   // sequencer 3: Empty Process
   INITIAL_STEP CheckMachineMode:   // S200, max time T#10S, warning time T#7S
   END_STEP
   TRANSITION Trans145 FROM CheckMachineMode TO WaitAllStoperReset   // T200
      := "AutoProcessControl".Global.K.EmptyPallet;
   END_TRANSITION
   STEP Step153:   // S153, max time T#10S, warning time T#7S
   END_STEP
   TRANSITION Trans163 FROM Step153 TO "CheckMachine Mode_6"   // T163, jump
      := TRUE;
   END_TRANSITION
   STEP "Process Finish_8":   // S244, max time T#10S, warning time T#7S
   END_STEP
   TRANSITION Trans257 FROM "Process Finish_8" TO Step153   // T256
      := TRUE;
   END_TRANSITION
   STEP LoadStop_14:   // S61, max time T#10S, warning time T#7S
   END_STEP
   TRANSITION Trans154 FROM LoadStop_14 TO CheckPalletExist_10   // T175
      := #LoadStop_14.T > t#2S;
   END_TRANSITION
   STEP LoadStop_12:   // S62, max time T#10S, warning time T#7S
   END_STEP
   TRANSITION Trans152 FROM LoadStop_12 TO CheckPalletExist_8   // T169
      := #LoadStop_12.T > t#2S;
   END_TRANSITION
   STEP "CheckMachine Mode_5":   // S158, max time T#10S, warning time T#7S
   END_STEP
   TRANSITION Trans175 FROM "CheckMachine Mode_5" TO LoadStop_13   // T196
      := "AutoProcessControl".Global.K.EmptyPallet;
   END_TRANSITION
   STEP LoadStop_13:   // S63, max time T#10S, warning time T#7S
   END_STEP
   TRANSITION Trans153 FROM LoadStop_13 TO CheckPalletExist_9   // T170
      := #LoadStop_13.T > t#2S;
   END_TRANSITION
   STEP CheckPalletExist_7:   // S64, max time T#10S, warning time T#7S
   END_STEP
   TRANSITION Trans66 FROM CheckPalletExist_7 TO WaitLineMotorReady_7   // T65
      := "K-reservePalletEmptyCheck1" AND (#CheckPalletExist_7.T > t#1000MS);
   END_TRANSITION
   TRANSITION Trans33 FROM CheckPalletExist_7 TO WaitPalletArive_9   // T32
      := NOT "K-reservePalletEmptyCheck1" AND (#CheckPalletExist_7.T > t#1000MS);
   END_TRANSITION
   STEP AriveTimeDelay_8:   // S159, max time T#10S, warning time T#7S
   END_STEP
   TRANSITION Trans151 FROM AriveTimeDelay_8 TO StoperReset_8   // T168
      := #AriveTimeDelay_8.T > t#500MS;
   END_TRANSITION
   STEP WaitLineMotorReady_7:   // S65, max time T#10S, warning time T#7S
   END_STEP
   TRANSITION Trans67 FROM WaitLineMotorReady_7 TO WaitPalletRequestRelease_7   // T66
      := "MotorControl".Dev[15].OutControl.o_Ready;
   END_TRANSITION
   STEP WaitPalletRequestRelease_7:   // S66, max time T#10S, warning time T#7S
   END_STEP
   TRANSITION Trans68 FROM WaitPalletRequestRelease_7 TO StoperRelease_8   // T67
      := NOT "iK-reserveTakeGateDetection";
   END_TRANSITION
   STEP LoadStop_11:   // S160, max time T#10S, warning time T#7S
   END_STEP
   TRANSITION Trans781 FROM LoadStop_11 TO CheckPalletExist_7   // T172
      := #LoadStop_11.T > t#2S;
   END_TRANSITION
   STEP WaitPalletArrveNextPos_7:   // S67, max time T#10S, warning time T#7S
   END_STEP
   TRANSITION Trans65 FROM WaitPalletArrveNextPos_7 TO AriveTimeDelay_8   // T64
      := "iK-reserveTakeGateDetection" OR NOT "AutoProcessControl".Global.K.EmptyPallet;
   END_TRANSITION
   STEP "Process Finish_9":   // S245, max time T#10S, warning time T#7S
   END_STEP
   TRANSITION Trans258 FROM "Process Finish_9" TO "CheckMachine Mode_7"   // T257, jump
      := TRUE;
   END_TRANSITION
   STEP StoperReset_8:   // S161, max time T#10S, warning time T#7S
              S    "ST10Cylinder".Cy[43].Inout.AutoGoHome
              R    "ST10Cylinder".Cy[43].Inout.AutoGoWork
   END_STEP
   TRANSITION Trans782 FROM StoperReset_8 TO "Process Finish_8"   // T173
      := TRUE;
   END_TRANSITION
   STEP StoperRelease_8:   // S162, max time T#10S, warning time T#7S
              R    "ST10Cylinder".Cy[43].Inout.AutoGoHome
              S    "ST10Cylinder".Cy[43].Inout.AutoGoWork
   END_STEP
   TRANSITION Trans783 FROM StoperRelease_8 TO WaitPalletArrveNextPos_7   // T174
      := #StoperRelease_8.T > t#1000MS;
   END_TRANSITION
   STEP CheckPalletExist_8:   // S68, max time T#10S, warning time T#7S
   END_STEP
   TRANSITION Trans70 FROM CheckPalletExist_8 TO WaitLineMotorReady_8   // T69
      := "K-reservePalletEmptyCheck2" AND (#CheckPalletExist_8.T > t#1000MS);
   END_TRANSITION
   TRANSITION Trans156 FROM CheckPalletExist_8 TO WaitPalletArive_6   // T179
      := NOT "K-reservePalletEmptyCheck2" AND (#CheckPalletExist_8.T > t#1000MS);
   END_TRANSITION
   STEP AriveTimeDelay_9:   // S163, max time T#10S, warning time T#7S
   END_STEP
   TRANSITION Trans155 FROM AriveTimeDelay_9 TO StoperReset_9   // T176
      := #AriveTimeDelay_9.T > t#500MS;
   END_TRANSITION
   STEP WaitLineMotorReady_8:   // S69, max time T#10S, warning time T#7S
   END_STEP
   TRANSITION Trans71 FROM WaitLineMotorReady_8 TO WaitPalletRequestRelease_8   // T70
      := "MotorControl".Dev[15].OutControl.o_Ready;
   END_TRANSITION
   STEP WaitPalletRequestRelease_8:   // S70, max time T#10S, warning time T#7S
   END_STEP
   TRANSITION Trans72 FROM WaitPalletRequestRelease_8 TO StoperRelease_9   // T71
      := "AutoProcessControl".Global.K.LoadStopRequestPallet_2;
   END_TRANSITION
   STEP WaitPalletArrveNextPos_8:   // S71, max time T#10S, warning time T#7S
   END_STEP
   TRANSITION Trans69 FROM WaitPalletArrveNextPos_8 TO AriveTimeDelay_9   // T68
      := "K-reservePalletEmptyCheck1";
   END_TRANSITION
   STEP StoperReset_9:   // S164, max time T#10S, warning time T#7S
              S    "ST10Cylinder".Cy[44].Inout.AutoGoHome
              R    "ST10Cylinder".Cy[44].Inout.AutoGoWork
   END_STEP
   TRANSITION Trans784 FROM StoperReset_9 TO "Process Finish_9"   // T177
      := TRUE;
   END_TRANSITION
   STEP StoperRelease_9:   // S165, max time T#10S, warning time T#7S
              R    "ST10Cylinder".Cy[44].Inout.AutoGoHome
              S    "ST10Cylinder".Cy[44].Inout.AutoGoWork
   END_STEP
   TRANSITION Trans785 FROM StoperRelease_9 TO WaitPalletArrveNextPos_8   // T178
      := #StoperRelease_9.T > t#1000MS;
   END_TRANSITION
   STEP WaitPalletArive_6:   // S166, max time T#10S, warning time T#7S
              N    "AutoProcessControl".Global.K.LoadStopRequestPallet_3
   END_STEP
   TRANSITION Trans157 FROM WaitPalletArive_6 TO TimeDelay_6   // T180
      := "K-reservePalletEmptyCheck2" OR NOT "AutoProcessControl".Global.K.EmptyPallet;
   END_TRANSITION
   STEP TimeDelay_6:   // S167, max time T#10S, warning time T#7S
   END_STEP
   TRANSITION Trans158 FROM TimeDelay_6 TO "CheckMachine Mode_7"   // T181, jump
      := #TimeDelay_6.T > t#500MS;
   END_TRANSITION
   STEP "Process Finish_10":   // S246, max time T#10S, warning time T#7S
   END_STEP
   TRANSITION Trans259 FROM "Process Finish_10" TO "CheckMachine Mode_5"   // T258, jump
      := TRUE;
   END_TRANSITION
   STEP CheckPalletExist_9:   // S72, max time T#10S, warning time T#7S
   END_STEP
   TRANSITION Trans74 FROM CheckPalletExist_9 TO WaitLineMotorReady_9   // T73
      := "K-reservePalletEmptyCheck3" AND (#CheckPalletExist_9.T > t#1000MS);
   END_TRANSITION
   TRANSITION Trans160 FROM CheckPalletExist_9 TO WaitPalletArive_7   // T185
      := NOT "K-reservePalletEmptyCheck3" AND (#CheckPalletExist_9.T > t#1000MS);
   END_TRANSITION
   STEP AriveTimeDelay_10:   // S168, max time T#10S, warning time T#7S
   END_STEP
   TRANSITION Trans159 FROM AriveTimeDelay_10 TO StoperReset_10   // T182
      := #AriveTimeDelay_10.T > t#500MS;
   END_TRANSITION
   STEP WaitLineMotorReady_9:   // S73, max time T#10S, warning time T#7S
   END_STEP
   TRANSITION Trans75 FROM WaitLineMotorReady_9 TO WaitPalletRequestRelease_9   // T74
      := "MotorControl".Dev[15].OutControl.o_Ready;
   END_TRANSITION
   STEP WaitPalletRequestRelease_9:   // S74, max time T#10S, warning time T#7S
   END_STEP
   TRANSITION Trans76 FROM WaitPalletRequestRelease_9 TO StoperRelease_10   // T75
      := "AutoProcessControl".Global.K.LoadStopRequestPallet_3;
   END_TRANSITION
   STEP WaitPalletArrveNextPos_9:   // S75, max time T#10S, warning time T#7S
   END_STEP
   TRANSITION Trans73 FROM WaitPalletArrveNextPos_9 TO AriveTimeDelay_10   // T72
      := "K-reservePalletEmptyCheck2";
   END_TRANSITION
   STEP StoperReset_10:   // S169, max time T#10S, warning time T#7S
              S    "ST10Cylinder".Cy[45].Inout.AutoGoHome
              R    "ST10Cylinder".Cy[45].Inout.AutoGoWork
   END_STEP
   TRANSITION Trans786 FROM StoperReset_10 TO "Process Finish_10"   // T183
      := TRUE;
   END_TRANSITION
   STEP StoperRelease_10:   // S170, max time T#10S, warning time T#7S
              R    "ST10Cylinder".Cy[45].Inout.AutoGoHome
              S    "ST10Cylinder".Cy[45].Inout.AutoGoWork
   END_STEP
   TRANSITION Trans787 FROM StoperRelease_10 TO WaitPalletArrveNextPos_9   // T184
      := #StoperRelease_10.T > t#1000MS;
   END_TRANSITION
   STEP WaitPalletArive_7:   // S171, max time T#10S, warning time T#7S
              N    "AutoProcessControl".Global.K.LoadStopRequestPallet_4
   END_STEP
   TRANSITION Trans161 FROM WaitPalletArive_7 TO TimeDelay_7   // T186
      := "K-reservePalletEmptyCheck3" OR NOT "AutoProcessControl".Global.K.EmptyPallet;
   END_TRANSITION
   STEP TimeDelay_7:   // S172, max time T#10S, warning time T#7S
   END_STEP
   TRANSITION Trans162 FROM TimeDelay_7 TO "CheckMachine Mode_5"   // T187, jump
      := #TimeDelay_7.T > t#500MS;
   END_TRANSITION
   STEP "Process Finish_11":   // S247, max time T#10S, warning time T#7S
   END_STEP
   TRANSITION Trans260 FROM "Process Finish_11" TO "CheckMachine Mode_8"   // T259, jump
      := TRUE;
   END_TRANSITION
   STEP CheckPalletExist_10:   // S76, max time T#10S, warning time T#7S
   END_STEP
   TRANSITION Trans78 FROM CheckPalletExist_10 TO WaitLineMotorReady_10   // T77
      := "K-reservePalletEmptyCheck4" AND NOT "iK-reserveMiddleDetection" AND (#CheckPalletExist_10.T > t#1000MS);
   END_TRANSITION
   TRANSITION Trans170 FROM CheckPalletExist_10 TO WaitPalletArive_8   // T191
      := NOT "K-reservePalletEmptyCheck4" AND (#CheckPalletExist_10.T > t#1000MS);
   END_TRANSITION
   STEP AriveTimeDelay_11:   // S173, max time T#10S, warning time T#7S
   END_STEP
   TRANSITION Trans169 FROM AriveTimeDelay_11 TO StoperReset_11   // T188
      := #AriveTimeDelay_11.T > t#500MS;
   END_TRANSITION
   STEP WaitLineMotorReady_10:   // S77, max time T#10S, warning time T#7S
   END_STEP
   TRANSITION Trans79 FROM WaitLineMotorReady_10 TO WaitPalletRequestRelease_10   // T78
      := "MotorControl".Dev[15].OutControl.o_Ready;
   END_TRANSITION
   STEP WaitPalletRequestRelease_10:   // S78, max time T#10S, warning time T#7S
   END_STEP
   TRANSITION Trans80 FROM WaitPalletRequestRelease_10 TO StoperRelease_11   // T79
      := "AutoProcessControl".Global.K.LoadStopRequestPallet_4;
   END_TRANSITION
   STEP WaitPalletArrveNextPos_10:   // S79, max time T#10S, warning time T#7S
   END_STEP
   TRANSITION Trans77 FROM WaitPalletArrveNextPos_10 TO AriveTimeDelay_11   // T76
      := "K-reservePalletEmptyCheck3";
   END_TRANSITION
   STEP StoperReset_11:   // S174, max time T#10S, warning time T#7S
              S    "ST10Cylinder".Cy[46].Inout.AutoGoHome
              R    "ST10Cylinder".Cy[46].Inout.AutoGoWork
   END_STEP
   TRANSITION Trans788 FROM StoperReset_11 TO "Process Finish_11"   // T189
      := TRUE;
   END_TRANSITION
   STEP StoperRelease_11:   // S175, max time T#10S, warning time T#7S
              R    "ST10Cylinder".Cy[46].Inout.AutoGoHome
              S    "ST10Cylinder".Cy[46].Inout.AutoGoWork
   END_STEP
   TRANSITION Trans789 FROM StoperRelease_11 TO WaitPalletArrveNextPos_10   // T190
      := #StoperRelease_11.T > t#1000MS;
   END_TRANSITION
   STEP WaitPalletArive_8:   // S176, max time T#10S, warning time T#7S
   END_STEP
   TRANSITION Trans171 FROM WaitPalletArive_8 TO TimeDelay_8   // T192
      := ("K-reservePalletEmptyCheck4" AND NOT "iK-reserveMiddleDetection") OR NOT "AutoProcessControl".Global.K.EmptyPallet;
   END_TRANSITION
   STEP TimeDelay_8:   // S177, max time T#10S, warning time T#7S
   END_STEP
   TRANSITION Trans172 FROM TimeDelay_8 TO "CheckMachine Mode_8"   // T193, jump
      := #TimeDelay_8.T > t#500MS;
   END_TRANSITION
   STEP "CheckMachine Mode_6":   // S178, max time T#10S, warning time T#7S
   END_STEP
   TRANSITION Trans173 FROM "CheckMachine Mode_6" TO LoadStop_11   // T194
      := "AutoProcessControl".Global.K.EmptyPallet;
   END_TRANSITION
   STEP "CheckMachine Mode_7":   // S179, max time T#10S, warning time T#7S
   END_STEP
   TRANSITION Trans174 FROM "CheckMachine Mode_7" TO LoadStop_12   // T195
      := "AutoProcessControl".Global.K.EmptyPallet;
   END_TRANSITION
   STEP "CheckMachine Mode_8":   // S180, max time T#10S, warning time T#7S
   END_STEP
   TRANSITION Trans168 FROM "CheckMachine Mode_8" TO LoadStop_14   // T171
      := "AutoProcessControl".Global.K.EmptyPallet;
   END_TRANSITION
   STEP WaitAllStoperReset:   // S181, max time T#10S, warning time T#7S
   END_STEP
   TRANSITION Trans197 FROM WaitAllStoperReset TO MotorRun_1   // T197
      := "ST10Cylinder".Cy[43].Inout.AutoGoHome AND NOT "ST10Cylinder".Cy[43].Inout.AutoGoWork AND "ST10Cylinder".Cy[44].Inout.AutoGoHome AND NOT "ST10Cylinder".Cy[44].Inout.AutoGoWork AND "ST10Cylinder".Cy[45].Inout.AutoGoHome AND NOT "ST10Cylinder".Cy[45].Inout.AutoGoWork AND "ST10Cylinder".Cy[46].Inout.AutoGoHome AND NOT "ST10Cylinder".Cy[46].Inout.AutoGoWork;
   END_TRANSITION
   STEP Step182:   // S182, max time T#10S, warning time T#7S
   END_STEP
   TRANSITION Trans198 FROM Step182 TO ("CheckMachine Mode_7", "CheckMachine Mode_5", "CheckMachine Mode_8", "CheckMachine Mode_6")   // T198
      := TRUE;
   END_TRANSITION
   STEP MotorRun_1:   // S80, max time T#10S, warning time T#7S
              R    "MotorControl".Dev[15].Auto.Start
              S    "MotorControl".Dev[15].Auto.CCWStart
              S    "MotorControl".Dev[16].Auto.Start
              R    "MotorControl".Dev[16].Auto.CCWStart
   END_STEP
   TRANSITION Trans81 FROM MotorRun_1 TO Step182   // T80
      := TRUE;
   END_TRANSITION
   STEP WaitPalletArive_9:   // S183, max time T#10S, warning time T#7S
              N    "AutoProcessControl".Global.K.LoadStopRequestPallet_2
   END_STEP
   TRANSITION Trans176 FROM WaitPalletArive_9 TO TimeDelay_9   // T199
      := "K-reservePalletEmptyCheck1" OR NOT "AutoProcessControl".Global.K.EmptyPallet;
   END_TRANSITION
   STEP TimeDelay_9:   // S184, max time T#10S, warning time T#7S
   END_STEP
   TRANSITION Trans177 FROM TimeDelay_9 TO "CheckMachine Mode_6"   // T201, jump
      := #TimeDelay_9.T > t#500MS;
   END_TRANSITION

   // permanent post-instructions
   NETWORK 1
      #ioPM_Inface.StepNum := #RT_DATA.S_DISPLAY;
   NETWORK 2
      IF #iSysInface.Reset THEN #AlarmID := 0; END_IF;
   NETWORK 3
      #TON[10].TON(IN := #工件放行中, PT := T#0.5S);
      IF #TON[10].Q THEN #工件放行中 := FALSE; END_IF;
END_FUNCTION_BLOCK

FUNCTION "ST10Cyl_interface91-100" : Void   // FC1029, LAD
{ S7_Optimized_Access := 'FALSE' }
// stored: AutoNumber false, SetENOAutomatically false
   VAR_INPUT
      AlwaysON : Bool;
      E_stop : Bool;
   END_VAR
   VAR_TEMP
      tTest : Bool;
   END_VAR
BEGIN

REGION Network 1 (SCL): Cylinder 91-100 IO Interface (SCL)
END_REGION

REGION Network 2: CY91 interface
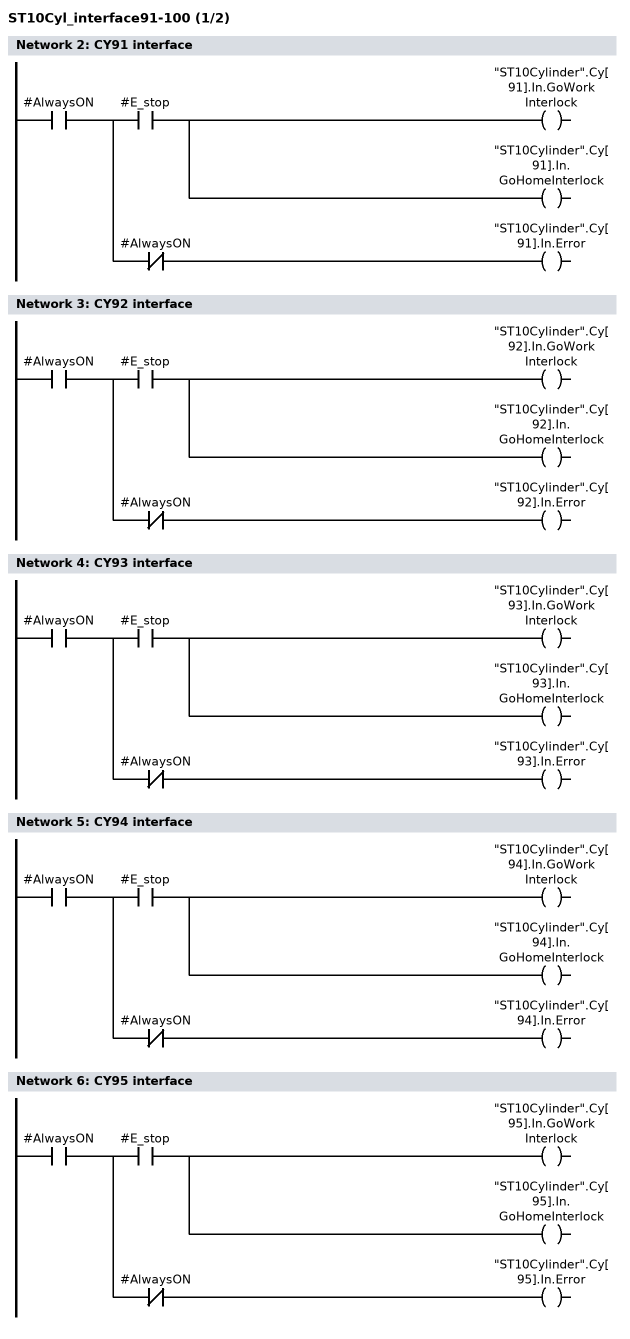
   RUNG wire#powerrail
      Contact( #AlwaysON )
      wire#w1
      Contact( #E_stop )
      wire#w2
      Coil( "ST10Cylinder".Cy[91].In.GoWorkInterlock )
   END_RUNG
   RUNG wire#w2
      Coil( "ST10Cylinder".Cy[91].In.GoHomeInterlock )
   END_RUNG
   RUNG wire#w1
      I_Contact( #AlwaysON )
      Coil( "ST10Cylinder".Cy[91].In.Error )
   END_RUNG
   // the same network as SCL:
   "ST10Cylinder".Cy[91].In.GoWorkInterlock := #AlwaysON AND #E_stop;
   "ST10Cylinder".Cy[91].In.GoHomeInterlock := #AlwaysON AND #E_stop;
   "ST10Cylinder".Cy[91].In.Error := #AlwaysON AND NOT #AlwaysON;
END_REGION

REGION Network 3: CY92 interface
   RUNG wire#powerrail
      Contact( #AlwaysON )
      wire#w1
      Contact( #E_stop )
      wire#w2
      Coil( "ST10Cylinder".Cy[92].In.GoWorkInterlock )
   END_RUNG
   RUNG wire#w2
      Coil( "ST10Cylinder".Cy[92].In.GoHomeInterlock )
   END_RUNG
   RUNG wire#w1
      I_Contact( #AlwaysON )
      Coil( "ST10Cylinder".Cy[92].In.Error )
   END_RUNG
   // the same network as SCL:
   "ST10Cylinder".Cy[92].In.GoWorkInterlock := #AlwaysON AND #E_stop;
   "ST10Cylinder".Cy[92].In.GoHomeInterlock := #AlwaysON AND #E_stop;
   "ST10Cylinder".Cy[92].In.Error := #AlwaysON AND NOT #AlwaysON;
END_REGION

REGION Network 4: CY93 interface
   RUNG wire#powerrail
      Contact( #AlwaysON )
      wire#w1
      Contact( #E_stop )
      wire#w2
      Coil( "ST10Cylinder".Cy[93].In.GoWorkInterlock )
   END_RUNG
   RUNG wire#w2
      Coil( "ST10Cylinder".Cy[93].In.GoHomeInterlock )
   END_RUNG
   RUNG wire#w1
      I_Contact( #AlwaysON )
      Coil( "ST10Cylinder".Cy[93].In.Error )
   END_RUNG
   // the same network as SCL:
   "ST10Cylinder".Cy[93].In.GoWorkInterlock := #AlwaysON AND #E_stop;
   "ST10Cylinder".Cy[93].In.GoHomeInterlock := #AlwaysON AND #E_stop;
   "ST10Cylinder".Cy[93].In.Error := #AlwaysON AND NOT #AlwaysON;
END_REGION

REGION Network 5: CY94 interface
   RUNG wire#powerrail
      Contact( #AlwaysON )
      wire#w1
      Contact( #E_stop )
      wire#w2
      Coil( "ST10Cylinder".Cy[94].In.GoWorkInterlock )
   END_RUNG
   RUNG wire#w2
      Coil( "ST10Cylinder".Cy[94].In.GoHomeInterlock )
   END_RUNG
   RUNG wire#w1
      I_Contact( #AlwaysON )
      Coil( "ST10Cylinder".Cy[94].In.Error )
   END_RUNG
   // the same network as SCL:
   "ST10Cylinder".Cy[94].In.GoWorkInterlock := #AlwaysON AND #E_stop;
   "ST10Cylinder".Cy[94].In.GoHomeInterlock := #AlwaysON AND #E_stop;
   "ST10Cylinder".Cy[94].In.Error := #AlwaysON AND NOT #AlwaysON;
END_REGION

REGION Network 6: CY95 interface
   RUNG wire#powerrail
      Contact( #AlwaysON )
      wire#w1
      Contact( #E_stop )
      wire#w2
      Coil( "ST10Cylinder".Cy[95].In.GoWorkInterlock )
   END_RUNG
   RUNG wire#w2
      Coil( "ST10Cylinder".Cy[95].In.GoHomeInterlock )
   END_RUNG
   RUNG wire#w1
      I_Contact( #AlwaysON )
      Coil( "ST10Cylinder".Cy[95].In.Error )
   END_RUNG
   // the same network as SCL:
   "ST10Cylinder".Cy[95].In.GoWorkInterlock := #AlwaysON AND #E_stop;
   "ST10Cylinder".Cy[95].In.GoHomeInterlock := #AlwaysON AND #E_stop;
   "ST10Cylinder".Cy[95].In.Error := #AlwaysON AND NOT #AlwaysON;
END_REGION

REGION Network 7: CY96 interface
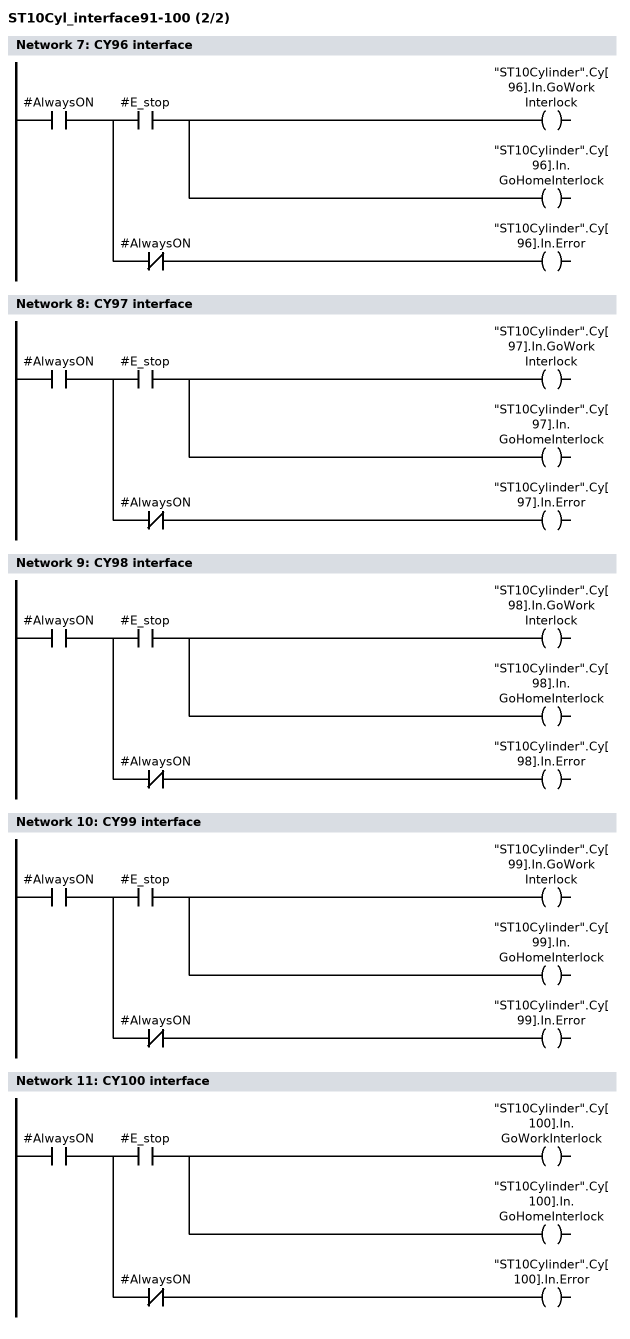
   RUNG wire#powerrail
      Contact( #AlwaysON )
      wire#w1
      Contact( #E_stop )
      wire#w2
      Coil( "ST10Cylinder".Cy[96].In.GoWorkInterlock )
   END_RUNG
   RUNG wire#w2
      Coil( "ST10Cylinder".Cy[96].In.GoHomeInterlock )
   END_RUNG
   RUNG wire#w1
      I_Contact( #AlwaysON )
      Coil( "ST10Cylinder".Cy[96].In.Error )
   END_RUNG
   // the same network as SCL:
   "ST10Cylinder".Cy[96].In.GoWorkInterlock := #AlwaysON AND #E_stop;
   "ST10Cylinder".Cy[96].In.GoHomeInterlock := #AlwaysON AND #E_stop;
   "ST10Cylinder".Cy[96].In.Error := #AlwaysON AND NOT #AlwaysON;
END_REGION

REGION Network 8: CY97 interface
   RUNG wire#powerrail
      Contact( #AlwaysON )
      wire#w1
      Contact( #E_stop )
      wire#w2
      Coil( "ST10Cylinder".Cy[97].In.GoWorkInterlock )
   END_RUNG
   RUNG wire#w2
      Coil( "ST10Cylinder".Cy[97].In.GoHomeInterlock )
   END_RUNG
   RUNG wire#w1
      I_Contact( #AlwaysON )
      Coil( "ST10Cylinder".Cy[97].In.Error )
   END_RUNG
   // the same network as SCL:
   "ST10Cylinder".Cy[97].In.GoWorkInterlock := #AlwaysON AND #E_stop;
   "ST10Cylinder".Cy[97].In.GoHomeInterlock := #AlwaysON AND #E_stop;
   "ST10Cylinder".Cy[97].In.Error := #AlwaysON AND NOT #AlwaysON;
END_REGION

REGION Network 9: CY98 interface
   RUNG wire#powerrail
      Contact( #AlwaysON )
      wire#w1
      Contact( #E_stop )
      wire#w2
      Coil( "ST10Cylinder".Cy[98].In.GoWorkInterlock )
   END_RUNG
   RUNG wire#w2
      Coil( "ST10Cylinder".Cy[98].In.GoHomeInterlock )
   END_RUNG
   RUNG wire#w1
      I_Contact( #AlwaysON )
      Coil( "ST10Cylinder".Cy[98].In.Error )
   END_RUNG
   // the same network as SCL:
   "ST10Cylinder".Cy[98].In.GoWorkInterlock := #AlwaysON AND #E_stop;
   "ST10Cylinder".Cy[98].In.GoHomeInterlock := #AlwaysON AND #E_stop;
   "ST10Cylinder".Cy[98].In.Error := #AlwaysON AND NOT #AlwaysON;
END_REGION

REGION Network 10: CY99 interface
   RUNG wire#powerrail
      Contact( #AlwaysON )
      wire#w1
      Contact( #E_stop )
      wire#w2
      Coil( "ST10Cylinder".Cy[99].In.GoWorkInterlock )
   END_RUNG
   RUNG wire#w2
      Coil( "ST10Cylinder".Cy[99].In.GoHomeInterlock )
   END_RUNG
   RUNG wire#w1
      I_Contact( #AlwaysON )
      Coil( "ST10Cylinder".Cy[99].In.Error )
   END_RUNG
   // the same network as SCL:
   "ST10Cylinder".Cy[99].In.GoWorkInterlock := #AlwaysON AND #E_stop;
   "ST10Cylinder".Cy[99].In.GoHomeInterlock := #AlwaysON AND #E_stop;
   "ST10Cylinder".Cy[99].In.Error := #AlwaysON AND NOT #AlwaysON;
END_REGION

REGION Network 11: CY100 interface
   RUNG wire#powerrail
      Contact( #AlwaysON )
      wire#w1
      Contact( #E_stop )
      wire#w2
      Coil( "ST10Cylinder".Cy[100].In.GoWorkInterlock )
   END_RUNG
   RUNG wire#w2
      Coil( "ST10Cylinder".Cy[100].In.GoHomeInterlock )
   END_RUNG
   RUNG wire#w1
      I_Contact( #AlwaysON )
      Coil( "ST10Cylinder".Cy[100].In.Error )
   END_RUNG
   // the same network as SCL:
   "ST10Cylinder".Cy[100].In.GoWorkInterlock := #AlwaysON AND #E_stop;
   "ST10Cylinder".Cy[100].In.GoHomeInterlock := #AlwaysON AND #E_stop;
   "ST10Cylinder".Cy[100].In.Error := #AlwaysON AND NOT #AlwaysON;
END_REGION
END_FUNCTION

FUNCTION_BLOCK "ST10_Stopper_FB"   // FB1160, LAD
{ S7_Optimized_Access := 'TRUE' }
// stored: AutoNumber false, MemoryReserve 100, SetENOAutomatically false
   VAR
      FB_Stopper_Instance { S7_SetPoint := 'True'} : Array[1..3] of "FB_Stopper";
   END_VAR
BEGIN

REGION Network 1 (SCL): A-托盘缓存阻挡气缸
       (*  
       REGION 允许释放条件,根据实际完善
           //马达运行中且工位一允许进料
           IF "ST350_Motor_InterfaceDB".aDev[1].Run  THEN
               "ST350_Stopper_InterfaceDB".Command[1].In.iReleaseClear := TRUE;
           ELSE
               "ST350_Stopper_InterfaceDB".Command[1].In.iReleaseClear := FALSE;
           END_IF;
       END_REGION

       REGION IO_image
           //InPut
           "ST350_Stopper_InterfaceDB".Command[1].In.iSensor := "iBurfferPalletDetection";//本站托盘到位
           "ST350_Stopper_InterfaceDB".Command[1].In.iNextSensor := "iWork01PalletDetection";//后站托盘到位
           "ST350_Stopper_InterfaceDB".Command[1].In.iNextValve := "oA-Lifting-01StopperCylinder";//后站挡停输出

           // //OutPut
            "ST10Cylinder".Cy[5].Inout.AutoGoWork:= "ST350_Stopper_InterfaceDB".Command[1].Out.oValve;//本站挡停输出
       END_REGION


       *)
END_REGION

REGION Network 2: #FB_Stopper_Instance[1] A-托盘缓存阻挡气缸
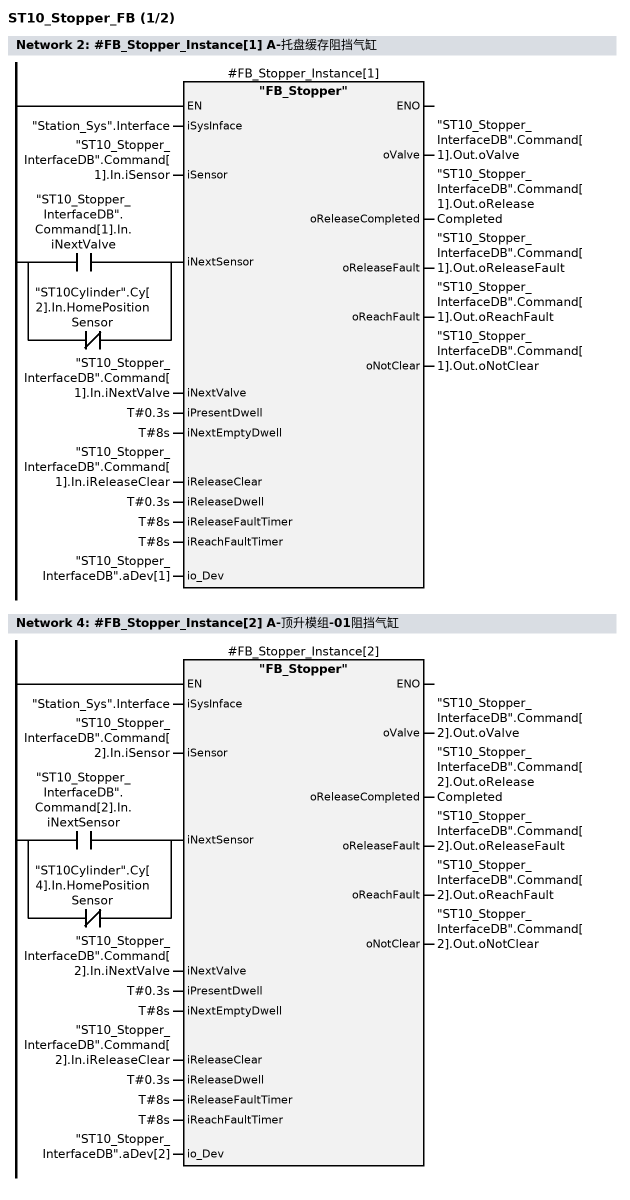
   RUNG wire#powerrail
      #FB_Stopper_Instance[1](iNextSensor := wire#w1, iSysInface := "Station_Sys".Interface, iSensor := "ST10_Stopper_InterfaceDB".Command[1].In.iSensor, iNextValve := "ST10_Stopper_InterfaceDB".Command[1].In.iNextValve, iPresentDwell := T#0.3s, iNextEmptyDwell := T#8s, iReleaseClear := "ST10_Stopper_InterfaceDB".Command[1].In.iReleaseClear, iReleaseDwell := T#0.3s, iReleaseFaultTimer := T#8s, iReachFaultTimer := T#8s, io_Dev := "ST10_Stopper_InterfaceDB".aDev[1], oValve => "ST10_Stopper_InterfaceDB".Command[1].Out.oValve, oReleaseCompleted => "ST10_Stopper_InterfaceDB".Command[1].Out.oReleaseCompleted, oReleaseFault => "ST10_Stopper_InterfaceDB".Command[1].Out.oReleaseFault, oReachFault => "ST10_Stopper_InterfaceDB".Command[1].Out.oReachFault, oNotClear => "ST10_Stopper_InterfaceDB".Command[1].Out.oNotClear)
   END_RUNG
   RUNG wire#powerrail
      Contact( "ST10_Stopper_InterfaceDB".Command[1].In.iNextValve )
   END_RUNG wire#w1
   RUNG wire#powerrail
      I_Contact( "ST10Cylinder".Cy[2].In.HomePositionSensor )
   END_RUNG wire#w1
   // the same network as SCL:
   #FB_Stopper_Instance[1](iSysInface := "Station_Sys".Interface,   // "FB_Stopper"
                           iSensor := "ST10_Stopper_InterfaceDB".Command[1].In.iSensor,
                           iNextSensor := "ST10_Stopper_InterfaceDB".Command[1].In.iNextValve OR NOT "ST10Cylinder".Cy[2].In.HomePositionSensor,
                           iNextValve := "ST10_Stopper_InterfaceDB".Command[1].In.iNextValve,
                           iPresentDwell := T#0.3s,
                           iNextEmptyDwell := T#8s,
                           iReleaseClear := "ST10_Stopper_InterfaceDB".Command[1].In.iReleaseClear,
                           iReleaseDwell := T#0.3s,
                           iReleaseFaultTimer := T#8s,
                           iReachFaultTimer := T#8s,
                           io_Dev := "ST10_Stopper_InterfaceDB".aDev[1],
                           oValve => "ST10_Stopper_InterfaceDB".Command[1].Out.oValve,
                           oReleaseCompleted => "ST10_Stopper_InterfaceDB".Command[1].Out.oReleaseCompleted,
                           oReleaseFault => "ST10_Stopper_InterfaceDB".Command[1].Out.oReleaseFault,
                           oReachFault => "ST10_Stopper_InterfaceDB".Command[1].Out.oReachFault,
                           oNotClear => "ST10_Stopper_InterfaceDB".Command[1].Out.oNotClear);
END_REGION

REGION Network 3 (SCL): A-顶升模组-01阻挡气缸
   (*
   REGION 允许释放条件,根据实际完善:顶升下降且线体运行中
       IF "ST10Cylinder".Cy[2].In.HomePositionSensor AND ("ST350_Motor_InterfaceDB".aDev[1].Run OR "Station_Sys".Manual.Mode) THEN//
           "ST350_Stopper_InterfaceDB".Command[2].In.iReleaseClear := True;
       ELSE
           "ST350_Stopper_InterfaceDB".Command[2].In.iReleaseClear := FALSE;
       END_IF;
   END_REGION

   REGION IO_image
       //InPut
       "ST350_Stopper_InterfaceDB".Command[2].In.iSensor := "iWork01PalletDetection";//本站托盘到位
       "ST350_Stopper_InterfaceDB".Command[2].In.iNextSensor := "iWork02PalletDetection";//后站托盘到位
       "ST350_Stopper_InterfaceDB".Command[2].In.iNextValve := "oA-Lifting-02StopperCylinder";//后站挡停输出

       // //OutPut
        "ST10Cylinder".Cy[1].Inout.AutoGoWork:= "ST350_Stopper_InterfaceDB".Command[2].Out.oValve;//本站挡停输出
   END_REGION

   *0
END_REGION

REGION Network 4: #FB_Stopper_Instance[2] A-顶升模组-01阻挡气缸
   RUNG wire#powerrail
      #FB_Stopper_Instance[2](iNextSensor := wire#w1, iSysInface := "Station_Sys".Interface, iSensor := "ST10_Stopper_InterfaceDB".Command[2].In.iSensor, iNextValve := "ST10_Stopper_InterfaceDB".Command[2].In.iNextValve, iPresentDwell := T#0.3s, iNextEmptyDwell := T#8s, iReleaseClear := "ST10_Stopper_InterfaceDB".Command[2].In.iReleaseClear, iReleaseDwell := T#0.3s, iReleaseFaultTimer := T#8s, iReachFaultTimer := T#8s, io_Dev := "ST10_Stopper_InterfaceDB".aDev[2], oValve => "ST10_Stopper_InterfaceDB".Command[2].Out.oValve, oReleaseCompleted => "ST10_Stopper_InterfaceDB".Command[2].Out.oReleaseCompleted, oReleaseFault => "ST10_Stopper_InterfaceDB".Command[2].Out.oReleaseFault, oReachFault => "ST10_Stopper_InterfaceDB".Command[2].Out.oReachFault, oNotClear => "ST10_Stopper_InterfaceDB".Command[2].Out.oNotClear)
   END_RUNG
   RUNG wire#powerrail
      Contact( "ST10_Stopper_InterfaceDB".Command[2].In.iNextSensor )
   END_RUNG wire#w1
   RUNG wire#powerrail
      I_Contact( "ST10Cylinder".Cy[4].In.HomePositionSensor )
   END_RUNG wire#w1
   // the same network as SCL:
   #FB_Stopper_Instance[2](iSysInface := "Station_Sys".Interface,   // "FB_Stopper"
                           iSensor := "ST10_Stopper_InterfaceDB".Command[2].In.iSensor,
                           iNextSensor := "ST10_Stopper_InterfaceDB".Command[2].In.iNextSensor OR NOT "ST10Cylinder".Cy[4].In.HomePositionSensor,
                           iNextValve := "ST10_Stopper_InterfaceDB".Command[2].In.iNextValve,
                           iPresentDwell := T#0.3s,
                           iNextEmptyDwell := T#8s,
                           iReleaseClear := "ST10_Stopper_InterfaceDB".Command[2].In.iReleaseClear,
                           iReleaseDwell := T#0.3s,
                           iReleaseFaultTimer := T#8s,
                           iReachFaultTimer := T#8s,
                           io_Dev := "ST10_Stopper_InterfaceDB".aDev[2],
                           oValve => "ST10_Stopper_InterfaceDB".Command[2].Out.oValve,
                           oReleaseCompleted => "ST10_Stopper_InterfaceDB".Command[2].Out.oReleaseCompleted,
                           oReleaseFault => "ST10_Stopper_InterfaceDB".Command[2].Out.oReleaseFault,
                           oReachFault => "ST10_Stopper_InterfaceDB".Command[2].Out.oReachFault,
                           oNotClear => "ST10_Stopper_InterfaceDB".Command[2].Out.oNotClear);
END_REGION

REGION Network 5 (SCL): A-顶升模组-02阻挡气缸
   //允许释放条件,根据实际完善:顶升下降且线体运行中
   (*

   REGION IOimage
       //InPut
       "ST350_Stopper_InterfaceDB".Command[3].In.iSensor := "iWork02PalletDetection";//本站托盘到位
       "ST350_Stopper_InterfaceDB".Command[3].In.iNextSensor := "iD-LiftingDetection" AND NOT "iD-LiftingINDetection" ;//后站托盘到位

       //替换后站挡停释放信号：升降机在下&顶升下&无料&允许金托盘
       // "ST350_Stopper_InterfaceDB".Command[3].In.iNextValve := ;//后站挡停输出

       // //OutPut
        "ST10Cylinder".Cy[3].Inout.AutoGoWork := "ST350_Stopper_InterfaceDB".Command[3].Out.oValve;//本站挡停输出


   END_REGION

   *)
END_REGION

REGION Network 6: #FB_Stopper_Instance[3] A-顶升模组-02阻挡气缸
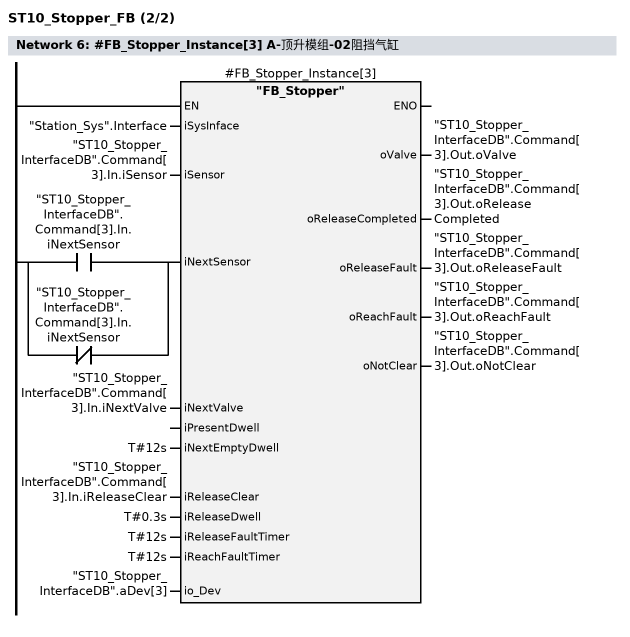
   RUNG wire#powerrail
      #FB_Stopper_Instance[3](iNextSensor := wire#w1, iSysInface := "Station_Sys".Interface, iSensor := "ST10_Stopper_InterfaceDB".Command[3].In.iSensor, iNextValve := "ST10_Stopper_InterfaceDB".Command[3].In.iNextValve, iPresentDwell :=, iNextEmptyDwell := T#12s, iReleaseClear := "ST10_Stopper_InterfaceDB".Command[3].In.iReleaseClear, iReleaseDwell := T#0.3s, iReleaseFaultTimer := T#12s, iReachFaultTimer := T#12s, io_Dev := "ST10_Stopper_InterfaceDB".aDev[3], oValve => "ST10_Stopper_InterfaceDB".Command[3].Out.oValve, oReleaseCompleted => "ST10_Stopper_InterfaceDB".Command[3].Out.oReleaseCompleted, oReleaseFault => "ST10_Stopper_InterfaceDB".Command[3].Out.oReleaseFault, oReachFault => "ST10_Stopper_InterfaceDB".Command[3].Out.oReachFault, oNotClear => "ST10_Stopper_InterfaceDB".Command[3].Out.oNotClear)
   END_RUNG
   RUNG wire#powerrail
      Contact( "ST10_Stopper_InterfaceDB".Command[3].In.iNextSensor )
   END_RUNG wire#w1
   RUNG wire#powerrail
      I_Contact( "ST10_Stopper_InterfaceDB".Command[3].In.iNextSensor )
   END_RUNG wire#w1
   // the same network as SCL:
   #FB_Stopper_Instance[3](iSysInface := "Station_Sys".Interface,   // "FB_Stopper"
                           iSensor := "ST10_Stopper_InterfaceDB".Command[3].In.iSensor,
                           iNextSensor := "ST10_Stopper_InterfaceDB".Command[3].In.iNextSensor OR NOT "ST10_Stopper_InterfaceDB".Command[3].In.iNextSensor,
                           iNextValve := "ST10_Stopper_InterfaceDB".Command[3].In.iNextValve,
                           iNextEmptyDwell := T#12s,
                           iReleaseClear := "ST10_Stopper_InterfaceDB".Command[3].In.iReleaseClear,
                           iReleaseDwell := T#0.3s,
                           iReleaseFaultTimer := T#12s,
                           iReachFaultTimer := T#12s,
                           io_Dev := "ST10_Stopper_InterfaceDB".aDev[3],
                           oValve => "ST10_Stopper_InterfaceDB".Command[3].Out.oValve,
                           oReleaseCompleted => "ST10_Stopper_InterfaceDB".Command[3].Out.oReleaseCompleted,
                           oReleaseFault => "ST10_Stopper_InterfaceDB".Command[3].Out.oReleaseFault,
                           oReachFault => "ST10_Stopper_InterfaceDB".Command[3].Out.oReachFault,
                           oNotClear => "ST10_Stopper_InterfaceDB".Command[3].Out.oNotClear);
END_REGION
END_FUNCTION_BLOCK

FUNCTION_BLOCK "SevroStart&PosCheck"   // FB4073, LAD
{ S7_Optimized_Access := 'TRUE' }
// stored: AutoNumber false, MemoryReserve 100, SetENOAutomatically false
   VAR_INPUT
      iRef_Homed { ExternalAccessible := 'False'; ExternalVisible := 'False'; ExternalWritable := 'False'} : Bool;
      iStandstill { ExternalAccessible := 'False'; ExternalVisible := 'False'; ExternalWritable := 'False'} : Bool;
      iReset : Bool;
      interlcok : Bool;   // 启动互锁
      "iActual Posi" { ExternalAccessible := 'False'; ExternalVisible := 'False'; ExternalWritable := 'False'} : DInt;
      "iTol+" { ExternalAccessible := 'False'; ExternalVisible := 'False'; ExternalWritable := 'False'} : DInt;
      "iTol-" { ExternalAccessible := 'False'; ExternalVisible := 'False'; ExternalWritable := 'False'} : DInt;
      iStartTon : Time := T#200ms;   // 启动延迟
   END_VAR
   VAR_OUTPUT
      oStartPos : Bool;   // 启动
      DoublePosError : Bool;   // 多位置触发
   END_VAR
   VAR_IN_OUT
      ioPoint : Array[0..39] of Struct
         Start : Bool;
         Achieve : Bool;
      END_STRUCT;
      ioList : "PosList";
      ioPosNumberSelect : Int;   // 位置启动
   END_VAR
   VAR
      TON : Array[0..1] of TON_TIME;
      StartCount { S7_SetPoint := 'True'} : Int;   // 启动计数
   END_VAR
   VAR_TEMP
      "Actual Posi+Tol" : DInt;
      "Actual Posi-Tol" : DInt;
      Index : Array[0..7] of Int;   // 位置启动
      PosStart : Bool;
   END_VAR
   VAR_TEMP   // added for the SCL form of the ladder/FBD networks
      _w1 : Bool;
   END_VAR
BEGIN

REGION Network 1 (SCL): 检查当前启动位置号
   #Index[1] := 0;
   #PosStart := false;
   FOR #Index[1] := 0 TO 39 DO
       IF #ioPoint[#Index[1]].Start THEN

           #ioPosNumberSelect := #Index[1];//当前启动位置号
           #PosStart := TRUE;
           EXIT;
       END_IF;
   END_FOR;
   #Index[2] := 0;
   #StartCount := 0;
   FOR #Index[2] := 0 TO 39 DO
       IF #ioPoint[#Index[2]].Start THEN

           #StartCount := #StartCount+1;//当前启动位置号


       END_IF;
       IF #Index[2] = 39 THEN

           EXIT;
       END_IF;

   END_FOR;
END_REGION

REGION Network 2: 位置给定
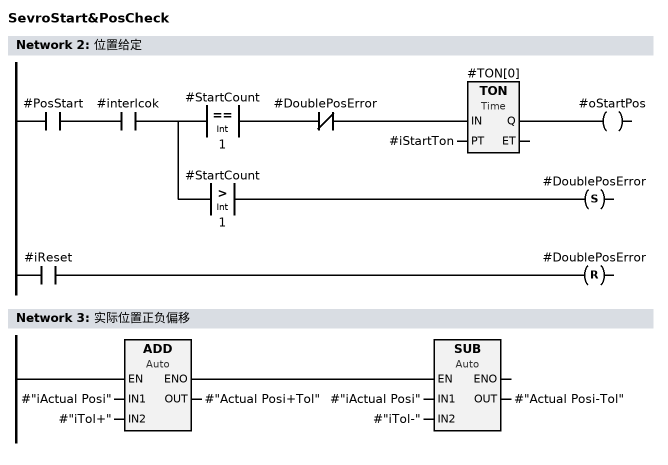
   RUNG wire#powerrail
      Contact( #PosStart )
      Contact( #interlcok )
      wire#w1
      { S7_Templates := "SrcType := Int" } EQ_Contact(in1 := #StartCount, in2 := 1)
      I_Contact( #DoublePosError )
      { S7_Templates := "time_type := Time" } #TON[0].TON(pt := #iStartTon, et =>)
      Coil( #oStartPos )
   END_RUNG
   RUNG wire#w1
      { S7_Templates := "SrcType := Int" } GT_Contact(in1 := #StartCount, in2 := 1)
      S_Coil( #DoublePosError )
   END_RUNG
   RUNG wire#powerrail
      Contact( #iReset )
      R_Coil( #DoublePosError )
   END_RUNG
   // the same network as SCL:
   #_w1 := #PosStart AND #interlcok;
   #TON[0].TON(IN := #_w1 AND (#StartCount = 1) AND NOT #DoublePosError, PT := #iStartTon);
   #oStartPos := #TON[0].Q;
   IF #_w1 AND (#StartCount > 1) THEN #DoublePosError := TRUE; END_IF;
   IF #iReset THEN #DoublePosError := FALSE; END_IF;
END_REGION

REGION Network 3: 实际位置正负偏移
   RUNG wire#powerrail
      Add(in1 := #"iActual Posi", in2 := #"iTol+", out => #"Actual Posi+Tol")
      Sub(in1 := #"iActual Posi", in2 := #"iTol-", out => #"Actual Posi-Tol")
   END_RUNG
   // the same network as SCL:
   #"Actual Posi+Tol" := #"iActual Posi" + #"iTol+";
   #"Actual Posi-Tol" := #"iActual Posi" - #"iTol-";
END_REGION

REGION Network 4 (SCL): 位置检查


   #Index[3] := 0;
   FOR #Index[3] := 0 TO 39 DO
       IF #ioList.List[ #Index[3]].Pos>= #"Actual Posi-Tol"
           AND #ioList.List[ #Index[3]].Pos<= #"Actual Posi+Tol"
       THEN
         #ioPoint[#Index[3]].Achieve := TRUE;
       ELSE
           #ioPoint[#Index[3]].Achieve := FALSE;
       END_IF;
   END_FOR;
END_REGION
END_FUNCTION_BLOCK

ORGANIZATION_BLOCK "07_CYCL_FLT"
{ S7_Optimized_Access := 'FALSE' }
VERSION : 0.1
   VAR_TEMP 
      OB80_EV_CLASS : Byte;
      OB80_FLT_ID : Byte;
      OB80_PRIORITY : Byte;
      OB80_OB_NUMBR : Byte;
      OB80_RESERVED_1 : Byte;
      OB80_RESERVED_2 : Byte;
      OB80_ERROR_INFO : Word;
      OB80_ERR_EV_CLASS : Byte;
      OB80_ERR_EV_NUM : Byte;
      OB80_OB_PRIORITY : Byte;
      OB80_OB_NUM : Byte;
      OB80_DATE_TIME : Date_And_Time;
   END_VAR


BEGIN
NETWORK
TITLE = 


END_ORGANIZATION_BLOCK

FUNCTION "ChangeOver" : Bool
{ S7_Optimized_Access := 'FALSE' }
AUTHOR : STD
FAMILY : RCS
VERSION : 18.0
   VAR_INPUT 
      iCheckType : String;
      "iPulse*500ms" : Bool;
      iReset : Bool;
   END_VAR

   VAR_OUTPUT 
      oPulse : Bool;
      oEqual : Bool;
   END_VAR

   VAR_IN_OUT 
      ioPreConfigType : String;
      ioCurrentName : String;
      iotime : Int;
      ioTrigger : Bool;
      ioPosEdg : Bool;
      ioAlarm : Bool;
      ioPls : Bool;
   END_VAR

   VAR_TEMP 
      tpPosEdg : Bool;
      tpPls : Bool;
   END_VAR


BEGIN
	//---------------------------------------------------------------//
	//FunctionName:ChangeOverV3
	//FunctionDescription:ChangeOver
	//---------------------------------------------------------------//
	(*in:
	
	iPreConfigType  String
	iLastType   String
	iPulse*500ms    Bool
	iTrigger    Bool
	
	
	//inout:
	//out:
	oPulse  Bool
	oAlarm  Bool
	
	*)
	//---------------------------------------------------------------//
	//Version:V2
	//D&T:2016-11-125
	//Group:RCS
	//Author:JM
	//-------------------------Modify1----------------------------------//
	//Version:V3.0
	//D&T:2016-11-28
	//Group: RCS
	//Author:JM
	//Modify: add timeout bit 
	//-------------------------Modify2----------------------------------//
	//Version:V3.0
	//D&T:20180416
	//Group: RCS
	//Author:JM
	//Modify:
	// Add pls flag in order to keep paramter that download after modifier safe.
	#tpPls := #ioTrigger AND NOT #ioPls;
	#ioPls := #ioTrigger;
	#tpPosEdg := #"iPulse*500ms" AND NOT #ioPosEdg;
	#ioPosEdg := #"iPulse*500ms";
	#oEqual := #ioPreConfigType = #iCheckType AND #ioPreConfigType<>'';
	
	
	// IF #tpPls THEN
	//     #ioPreConfigType:='';
	// END_IF;
	IF (#iReset AND #ioAlarm) OR #oEqual THEN
	    #ioAlarm := 0;
	END_IF;
	IF NOT #ioTrigger THEN
	    #ChangeOver := 0;
	    #iotime := 0;
	    // #oAlarm := 0;
	    RETURN;
	ELSE
	    IF #tpPosEdg THEN
	        #iotime := #iotime + 1;
	    END_IF;
	    IF #iotime >= 10 THEN
	        #ioAlarm := 1;
	        #ioTrigger := 0;
	        // ELSE
	        //     #oAlarm := 0;
	    END_IF;
	    #ChangeOver := 0;
	    // #tpCurrentProductlen := LEN(#tpCurrentProduct);
	    // #tpLastProductlen := LEN(#tpLastProduct);
	    IF #ioPreConfigType <> #iCheckType THEN
	        #oPulse := #"iPulse*500ms";
	        RETURN;
	    ELSE
	        IF #ioCurrentName <> #ioPreConfigType THEN
	            #ioCurrentName := #ioPreConfigType;
	        END_IF;
	        #iotime := 0;
	        #ioAlarm := 0;
	        #oPulse := 0;
	        #ChangeOver := 1;
	        #ioTrigger := 0;
	        ENO := 1;
	    END_IF;
	    
	END_IF;
	
END_FUNCTION

FUNCTION_BLOCK "FB_AteqF620"
{ S7_Optimized_Access := 'FALSE' }
AUTHOR : 'Chaoyao.Zheng'
FAMILY : LeakTester
VERSION : 1.0
   VAR_INPUT 
      iHWID_Slot1 { ExternalAccessible := 'False'; ExternalVisible := 'False'; ExternalWritable := 'False'} : HW_IO;
      iHWID_Slot2 { ExternalAccessible := 'False'; ExternalVisible := 'False'; ExternalWritable := 'False'} : HW_IO;
      iHWID_Slot3 { ExternalAccessible := 'False'; ExternalVisible := 'False'; ExternalWritable := 'False'} : HW_IO;
      iHWID_Slot4 { ExternalAccessible := 'False'; ExternalVisible := 'False'; ExternalWritable := 'False'} : HW_IO;
      iHWID_Slot5 { ExternalAccessible := 'False'; ExternalVisible := 'False'; ExternalWritable := 'False'} : HW_IO;
      iHWID_Slot6 { ExternalAccessible := 'False'; ExternalVisible := 'False'; ExternalWritable := 'False'} : HW_IO;
      iHWID_Slot7 { ExternalAccessible := 'False'; ExternalVisible := 'False'; ExternalWritable := 'False'} : HW_IO;
      iHWID_Slot8 { ExternalAccessible := 'False'; ExternalVisible := 'False'; ExternalWritable := 'False'} : HW_IO;
      iSysRun { ExternalAccessible := 'False'; ExternalVisible := 'False'; ExternalWritable := 'False'} : Bool;
      iReset { ExternalAccessible := 'False'; ExternalVisible := 'False'; ExternalWritable := 'False'} : Bool;
      iAuto { ExternalAccessible := 'False'; ExternalVisible := 'False'; ExternalWritable := 'False'} : Bool;
      iManual { ExternalAccessible := 'False'; ExternalVisible := 'False'; ExternalWritable := 'False'} : Bool;
      iTimeout { ExternalAccessible := 'False'; ExternalVisible := 'False'; ExternalWritable := 'False'} : Time := T#5S;
   END_VAR

   VAR_OUTPUT 
      oDeviceReady { ExternalAccessible := 'False'; ExternalVisible := 'False'; ExternalWritable := 'False'} : Bool;
      oReady { ExternalAccessible := 'False'; ExternalVisible := 'False'; ExternalWritable := 'False'} : Bool;
      oError { ExternalAccessible := 'False'; ExternalVisible := 'False'; ExternalWritable := 'False'} : Bool;
      oSetProgOk { ExternalAccessible := 'False'; ExternalVisible := 'False'; ExternalWritable := 'False'} : Bool;
      oMeasureOk { ExternalAccessible := 'False'; ExternalVisible := 'False'; ExternalWritable := 'False'} : Bool;
      oErrorCode { ExternalAccessible := 'False'; ExternalVisible := 'False'; ExternalWritable := 'False'} : UInt;
      oFillTime : Real;
      oStabTime : Real;
      oTeatTime : Real;
      oDumpTime : Real;
      oResult { ExternalAccessible := 'False'; ExternalVisible := 'False'; ExternalWritable := 'False'} : Struct
         PassPart { ExternalAccessible := 'False'; ExternalVisible := 'False'; ExternalWritable := 'False'} : Bool;
         FailTestPart { ExternalAccessible := 'False'; ExternalVisible := 'False'; ExternalWritable := 'False'} : Bool;
         FailRefPart { ExternalAccessible := 'False'; ExternalVisible := 'False'; ExternalWritable := 'False'} : Bool;
         Alarm { ExternalAccessible := 'False'; ExternalVisible := 'False'; ExternalWritable := 'False'} : Bool;
         PressureError { ExternalAccessible := 'False'; ExternalVisible := 'False'; ExternalWritable := 'False'} : Bool;
         PartRecoverable { ExternalAccessible := 'False'; ExternalVisible := 'False'; ExternalWritable := 'False'} : Bool;
         CalibError { ExternalAccessible := 'False'; ExternalVisible := 'False'; ExternalWritable := 'False'} : Bool;
         CalibCheckError { ExternalAccessible := 'False'; ExternalVisible := 'False'; ExternalWritable := 'False'} : Bool;
         AtrFault { ExternalAccessible := 'False'; ExternalVisible := 'False'; ExternalWritable := 'False'} : Bool;
         Leak { ExternalAccessible := 'False'; ExternalVisible := 'False'; ExternalWritable := 'False'} : Struct
            Value { ExternalAccessible := 'False'; ExternalVisible := 'False'; ExternalWritable := 'False'} : Real;
            Unit { ExternalAccessible := 'False'; ExternalVisible := 'False'; ExternalWritable := 'False'} : String[10];
         END_STRUCT;
      END_STRUCT;
      oPressure { ExternalAccessible := 'False'; ExternalVisible := 'False'; ExternalWritable := 'False'} : Struct
         Value { ExternalAccessible := 'False'; ExternalVisible := 'False'; ExternalWritable := 'False'} : Real;
         Unit { ExternalAccessible := 'False'; ExternalVisible := 'False'; ExternalWritable := 'False'} : String[10];
      END_STRUCT;
      oActProgStep { ExternalAccessible := 'False'; ExternalVisible := 'False'; ExternalWritable := 'False'} : UInt;
      oActProgNo { ExternalAccessible := 'False'; ExternalVisible := 'False'; ExternalWritable := 'False'} : UInt;
      oElapsedTime { ExternalAccessible := 'False'; ExternalVisible := 'False'; ExternalWritable := 'False'} : Time;
   END_VAR

   VAR_IN_OUT 
      ioSetProg { ExternalAccessible := 'False'; ExternalVisible := 'False'; ExternalWritable := 'False'} : Bool;
      ioMeasure { ExternalAccessible := 'False'; ExternalVisible := 'False'; ExternalWritable := 'False'} : Bool;
      ioSpecialCycle : Bool;
      ioReadProTime : Bool;
   END_VAR

   VAR 
      sHMI { S7_SetPoint := 'False'} : "RCS_typeAteqF620Visual";
      sAuto { ExternalAccessible := 'False'; ExternalVisible := 'False'; ExternalWritable := 'False'} : Struct
         Set { ExternalAccessible := 'False'; ExternalVisible := 'False'; ExternalWritable := 'False'} : Struct
            ProgNo { ExternalAccessible := 'False'; ExternalVisible := 'False'; ExternalWritable := 'False'} : UInt;
         END_STRUCT;
      END_STRUCT;
      sHelp { ExternalAccessible := 'False'; ExternalVisible := 'False'; ExternalWritable := 'False'} : Struct
         First { ExternalAccessible := 'False'; ExternalVisible := 'False'; ExternalWritable := 'False'} : Bool := FALSE;
         AutoOld { ExternalAccessible := 'False'; ExternalVisible := 'False'; ExternalWritable := 'False'} : Bool;
         ManualOld { ExternalAccessible := 'False'; ExternalVisible := 'False'; ExternalWritable := 'False'} : Bool;
         ResetRis { ExternalAccessible := 'False'; ExternalVisible := 'False'; ExternalWritable := 'False'} : Bool;
         ResetOld { ExternalAccessible := 'False'; ExternalVisible := 'False'; ExternalWritable := 'False'} : Bool;
         SetProgRis { ExternalAccessible := 'False'; ExternalVisible := 'False'; ExternalWritable := 'False'} : Bool;
         SetProgOld { ExternalAccessible := 'False'; ExternalVisible := 'False'; ExternalWritable := 'False'} : Bool;
         SetProgAct { ExternalAccessible := 'False'; ExternalVisible := 'False'; ExternalWritable := 'False'} : Bool;
         MeasureRis { ExternalAccessible := 'False'; ExternalVisible := 'False'; ExternalWritable := 'False'} : Bool;
         MeasureOld { ExternalAccessible := 'False'; ExternalVisible := 'False'; ExternalWritable := 'False'} : Bool;
         MeasureAct { ExternalAccessible := 'False'; ExternalVisible := 'False'; ExternalWritable := 'False'} : Bool;
         EnableTime { ExternalAccessible := 'False'; ExternalVisible := 'False'; ExternalWritable := 'False'} : Bool;
         Abort { ExternalAccessible := 'False'; ExternalVisible := 'False'; ExternalWritable := 'False'} : Bool;
         OrderCnt { ExternalAccessible := 'False'; ExternalVisible := 'False'; ExternalWritable := 'False'} : UInt;
         Step { ExternalAccessible := 'False'; ExternalVisible := 'False'; ExternalWritable := 'False'} : Array[1..2] of UInt;
         CmdTimer {InstructionName := 'TON_TIME'; LibVersion := '1.0'; ExternalAccessible := 'False'; ExternalVisible := 'False'; ExternalWritable := 'False'} : TON_TIME;
         Set { ExternalAccessible := 'False'; ExternalVisible := 'False'; ExternalWritable := 'False'} : Struct
            ProgNo { ExternalAccessible := 'False'; ExternalVisible := 'False'; ExternalWritable := 'False'} : UInt;
         END_STRUCT;
      END_STRUCT;
      sRecv { ExternalAccessible := 'False'; ExternalVisible := 'False'; ExternalWritable := 'False'} : Struct
         Echo { ExternalAccessible := 'False'; ExternalVisible := 'False'; ExternalWritable := 'False'} : Struct
            Reset { ExternalAccessible := 'False'; ExternalVisible := 'False'; ExternalWritable := 'False'} : Bool;
            Start { ExternalAccessible := 'False'; ExternalVisible := 'False'; ExternalWritable := 'False'} : Bool;
            StartSpec { ExternalAccessible := 'False'; ExternalVisible := 'False'; ExternalWritable := 'False'} : Bool;
            ProgramSel { ExternalAccessible := 'False'; ExternalVisible := 'False'; ExternalWritable := 'False'} : Bool;
            ReadPara { ExternalAccessible := 'False'; ExternalVisible := 'False'; ExternalWritable := 'False'} : Bool;
            ReadLastResult { ExternalAccessible := 'False'; ExternalVisible := 'False'; ExternalWritable := 'False'} : Bool;
            Status { ExternalAccessible := 'False'; ExternalVisible := 'False'; ExternalWritable := 'False'} : UInt;
         END_STRUCT;
         Result { ExternalAccessible := 'False'; ExternalVisible := 'False'; ExternalWritable := 'False'} : Struct
            PassPart { ExternalAccessible := 'False'; ExternalVisible := 'False'; ExternalWritable := 'False'} : Bool;
            FailTestPart { ExternalAccessible := 'False'; ExternalVisible := 'False'; ExternalWritable := 'False'} : Bool;
            FailRefPart { ExternalAccessible := 'False'; ExternalVisible := 'False'; ExternalWritable := 'False'} : Bool;
            Alarm { ExternalAccessible := 'False'; ExternalVisible := 'False'; ExternalWritable := 'False'} : Bool;
            PressureError { ExternalAccessible := 'False'; ExternalVisible := 'False'; ExternalWritable := 'False'} : Bool;
            PartRecoverable { ExternalAccessible := 'False'; ExternalVisible := 'False'; ExternalWritable := 'False'} : Bool;
            CalibError { ExternalAccessible := 'False'; ExternalVisible := 'False'; ExternalWritable := 'False'} : Bool;
            CalibCheckError { ExternalAccessible := 'False'; ExternalVisible := 'False'; ExternalWritable := 'False'} : Bool;
            AtrFault { ExternalAccessible := 'False'; ExternalVisible := 'False'; ExternalWritable := 'False'} : Bool;
            Leak { ExternalAccessible := 'False'; ExternalVisible := 'False'; ExternalWritable := 'False'} : Struct
               Value { ExternalAccessible := 'False'; ExternalVisible := 'False'; ExternalWritable := 'False'} : Real;
               Unit { ExternalAccessible := 'False'; ExternalVisible := 'False'; ExternalWritable := 'False'} : String[10];
            END_STRUCT;
         END_STRUCT;
         CycleEnd { ExternalAccessible := 'False'; ExternalVisible := 'False'; ExternalWritable := 'False'} : Bool;
         ErrorCode { ExternalAccessible := 'False'; ExternalVisible := 'False'; ExternalWritable := 'False'} : UInt;
         ActProgram { ExternalAccessible := 'False'; ExternalVisible := 'False'; ExternalWritable := 'False'} : UInt;
         ResultCnt { ExternalAccessible := 'False'; ExternalVisible := 'False'; ExternalWritable := 'False'} : UInt;
         ActTestType { ExternalAccessible := 'False'; ExternalVisible := 'False'; ExternalWritable := 'False'} : UInt;
         ActProgStep { ExternalAccessible := 'False'; ExternalVisible := 'False'; ExternalWritable := 'False'} : UInt;
         ActPressure { ExternalAccessible := 'False'; ExternalVisible := 'False'; ExternalWritable := 'False'} : UDInt;
         PressureUnitCode { ExternalAccessible := 'False'; ExternalVisible := 'False'; ExternalWritable := 'False'} : UDInt;
         ActLeak { ExternalAccessible := 'False'; ExternalVisible := 'False'; ExternalWritable := 'False'} : UDInt;
         LeakUnitCode { ExternalAccessible := 'False'; ExternalVisible := 'False'; ExternalWritable := 'False'} : UDInt;
         FillTime { ExternalAccessible := 'False'; ExternalVisible := 'False'; ExternalWritable := 'False'} : UDInt;
         StabTime { ExternalAccessible := 'False'; ExternalVisible := 'False'; ExternalWritable := 'False'} : UDInt;
         TeatTime { ExternalAccessible := 'False'; ExternalVisible := 'False'; ExternalWritable := 'False'} : UDInt;
         DumpTime { ExternalAccessible := 'False'; ExternalVisible := 'False'; ExternalWritable := 'False'} : UDInt;
      END_STRUCT;
      sSend { ExternalAccessible := 'False'; ExternalVisible := 'False'; ExternalWritable := 'False'} : Struct
         Reset { ExternalAccessible := 'False'; ExternalVisible := 'False'; ExternalWritable := 'False'} : Bool;
         Start { ExternalAccessible := 'False'; ExternalVisible := 'False'; ExternalWritable := 'False'} : Bool;
         StartSpec { ExternalAccessible := 'False'; ExternalVisible := 'False'; ExternalWritable := 'False'} : Bool;
         ProgramSel { ExternalAccessible := 'False'; ExternalVisible := 'False'; ExternalWritable := 'False'} : Bool;
         ReadPara { ExternalAccessible := 'False'; ExternalVisible := 'False'; ExternalWritable := 'False'} : Bool;
         ReadLastResult { ExternalAccessible := 'False'; ExternalVisible := 'False'; ExternalWritable := 'False'} : Bool;
         ProgNo { ExternalAccessible := 'False'; ExternalVisible := 'False'; ExternalWritable := 'False'} : UInt;
      END_STRUCT;
      sArrayInput { ExternalAccessible := 'False'; ExternalVisible := 'False'; ExternalWritable := 'False'} : Array[1..#cSlotAmount, 1..#cFieldbusBytes] of Byte;
      sArrayOutput { ExternalAccessible := 'False'; ExternalVisible := 'False'; ExternalWritable := 'False'} : Array[1..#cSlotAmount, 1..#cFieldbusBytes] of Byte;
      SpecialCycleStep : Int;
      ReadProTimeStep : Int;
      IEC_Timer_0_Instance {InstructionName := 'TON_TIME'; LibVersion := '1.0'} : TON_TIME;
      IEC_Timer_1_Instance {InstructionName := 'TON_TIME'; LibVersion := '1.0'} : TON_TIME;
      IEC_Timer_0_Instance_1 {InstructionName := 'TON_TIME'; LibVersion := '1.0'} : TON_TIME;
      IEC_Timer_1_Instance_1 {InstructionName := 'TON_TIME'; LibVersion := '1.0'} : TON_TIME;
      IEC_Timer_2_Instance_1 {InstructionName := 'TON_TIME'; LibVersion := '1.0'} : TON_TIME;
   END_VAR

   VAR_TEMP 
      tIndex : UInt;
      tLoop : Int;
      tZero : Byte;
      tRetval : Struct
         LocallyErrID : Word;
         DPRD : Array[1..#cSlotAmount] of Int;
         DPWR : Array[1..#cSlotAmount] of Int;
         FILL : Int;
      END_STRUCT;
   END_VAR

   VAR CONSTANT 
      cSlotAmount : UInt := 4;
      cFieldbusBytes : UInt := 64;
   END_VAR


BEGIN
	REGION Description header
	    //================================================================================
	    // (C) Ruhlamat Automation Technologies (Suzhou) Co.,Ltd.
	    //--------------------------------------------------------------------------------
	    // TargetSystem: ATEQ F620(COMX 100XX-PNS)
	    // Engineering : TIA Portal V15 SP1
	    // Author      : Chaoyao.Zheng
	    //--------------------------------------------------------------------------------
	    // Moduleversions:
	    // V1.0 2020-08-24 - Chaoyao
	    // - Initial version
	    //================================================================================
	END_REGION
	REGION Error code explanation
	    //  100: DPRD_DAT error occurred                                    
	    //  101: DPWR_DAT error occurred                                    
	    //  102: GET_ERR_ID error occurred                                  
	    //  200: Order while FB not ready (oReady=FALSE)                    
	    //  201: Several orders set at the same time                        
	    //  202: Program number is not valid (1-128)                        
	    //  203: Command error occurred                                     
	    //  204: Command timeout                                            
	END_REGION
	
	(* FB Init *)
	IF NOT #sHelp.First THEN
	    (* initialize outputs *)
	    #sHelp.Abort := FALSE;
	    #oDeviceReady := FALSE;
	    #oReady := FALSE;
	    #oSetProgOk := FALSE;
	    #oMeasureOk := FALSE;
	    #oErrorCode := 0;
	    #oElapsedTime := T#0s;
	    #tZero := 0;
	    #tRetval.FILL := FILL(BVAL := #tZero, BLK => #oResult);
	    #sHMI.Status.InstanceName := GetInstanceName(0);
	    #sHelp.First := TRUE;
	ELSE
	    (* reset fieldbus output *)
	    FOR #tLoop := 1 TO UINT_TO_INT(#cSlotAmount) DO
	        UFILL_BLK(IN := 0,
	                  COUNT := #cFieldbusBytes,
	                  OUT => #sArrayOutput[#tLoop, 01]);
	    END_FOR;
	    
	    (* cyclic read tester input *)
	    #tRetval.DPRD[1] := DPRD_DAT(LADDR := #iHWID_Slot1,
	                                 RECORD => #sArrayInput[1]);
	    #tRetval.DPRD[2] := DPRD_DAT(LADDR := #iHWID_Slot2,
	                                 RECORD => #sArrayInput[2]);
	    #tRetval.DPRD[3] := DPRD_DAT(LADDR := #iHWID_Slot3,
	                                 RECORD => #sArrayInput[3]);
	    #tRetval.DPRD[4] := DPRD_DAT(LADDR := #iHWID_Slot4,
	                                 RECORD => #sArrayInput[4]);
	    IF (#tRetval.DPRD[1] <> 0) OR (#tRetval.DPRD[2] <> 0) OR (#tRetval.DPRD[3] <> 0) OR (#tRetval.DPRD[4] <> 0) THEN
	        #oErrorCode := 100; // Error cyclic read
	    END_IF;
	    
	    (* move input bytes to static bits *)
	    #sRecv.Echo.Reset := #sArrayInput[1, 01].%X0;
	    #sRecv.Echo.Start := #sArrayInput[1, 01].%X1;
	    #sRecv.Echo.StartSpec := #sArrayInput[1, 01].%X2;
	    #sRecv.Echo.ProgramSel := #sArrayInput[1, 01].%X3;
	    #sRecv.Echo.ReadPara := #sArrayInput[1, 02].%X5;
	    #sRecv.Echo.ReadLastResult := #sArrayInput[1, 02].%X7;
	    #sRecv.Result.PassPart := #sArrayInput[1, 13].%X0;
	    #sRecv.Result.FailTestPart := #sArrayInput[1, 13].%X1;
	    #sRecv.Result.FailRefPart := #sArrayInput[1, 13].%X2;
	    #sRecv.Result.Alarm := #sArrayInput[1, 13].%X3;
	    #sRecv.Result.PressureError := #sArrayInput[1, 13].%X4;
	    #sRecv.CycleEnd := #sArrayInput[1, 13].%X5;
	    #sRecv.Result.PartRecoverable := #sArrayInput[1, 13].%X6;
	    #sRecv.Result.CalibError := #sArrayInput[1, 13].%X7;
	    #sRecv.Result.CalibCheckError := #sArrayInput[1, 14].%X0;
	    #sRecv.Result.AtrFault := #sArrayInput[1, 14].%X1;
	    #sRecv.Result.Leak.Value := DINT_TO_REAL(#sRecv.ActLeak) / 1000.0;
	    #oFillTime := DINT_TO_REAL(#sRecv.FillTime) / 1000.0;
	    #oStabTime := DINT_TO_REAL(#sRecv.StabTime) / 1000.0;
	    #oTeatTime := DINT_TO_REAL(#sRecv.TeatTime) / 1000.0;
	    #oDumpTime := DINT_TO_REAL(#sRecv.DumpTime) / 1000.0;
	    #sRecv.Echo.Status.%B0 := #sArrayInput[1, 01];
	    #sRecv.Echo.Status.%B1 := #sArrayInput[1, 02];
	    #sRecv.ErrorCode.%B0 := #sArrayInput[1, 03];
	    #sRecv.ErrorCode.%B1 := #sArrayInput[1, 04];
	    #sRecv.ActProgram.%B0 := #sArrayInput[1, 07];
	    #sRecv.ActProgram.%B1 := #sArrayInput[1, 08];
	    #sRecv.ActProgStep.%B0 := #sArrayInput[1, 15];
	    #sRecv.ActProgStep.%B1 := #sArrayInput[1, 16];
	    #sRecv.ActPressure.%B0 := #sArrayInput[1, 17];
	    #sRecv.ActPressure.%B1 := #sArrayInput[1, 18];
	    #sRecv.ActPressure.%B2 := #sArrayInput[1, 19];
	    #sRecv.ActPressure.%B3 := #sArrayInput[1, 20];
	    #sRecv.PressureUnitCode.%B0 := #sArrayInput[1, 21];
	    #sRecv.PressureUnitCode.%B1 := #sArrayInput[1, 22];
	    #sRecv.PressureUnitCode.%B2 := #sArrayInput[1, 23];
	    #sRecv.PressureUnitCode.%B3 := #sArrayInput[1, 24];
	    #sRecv.ActLeak.%B0 := #sArrayInput[1, 25];
	    #sRecv.ActLeak.%B1 := #sArrayInput[1, 26];
	    #sRecv.ActLeak.%B2 := #sArrayInput[1, 27];
	    #sRecv.ActLeak.%B3 := #sArrayInput[1, 28];
	    #sRecv.LeakUnitCode.%B0 := #sArrayInput[1, 29];
	    #sRecv.LeakUnitCode.%B1 := #sArrayInput[1, 30];
	    #sRecv.LeakUnitCode.%B2 := #sArrayInput[1, 31];
	    #sRecv.LeakUnitCode.%B3 := #sArrayInput[1, 32];
	    #sRecv.FillTime.%B0 := #sArrayInput[1, 35];
	    #sRecv.FillTime.%B1 := #sArrayInput[1, 36];
	    #sRecv.FillTime.%B2 := #sArrayInput[1, 37];
	    #sRecv.FillTime.%B3 := #sArrayInput[1, 38];
	    #sRecv.StabTime.%B0 := #sArrayInput[1, 41];
	    #sRecv.StabTime.%B1 := #sArrayInput[1, 42];
	    #sRecv.StabTime.%B2 := #sArrayInput[1, 43];
	    #sRecv.StabTime.%B3 := #sArrayInput[1, 44];
	    #sRecv.TeatTime.%B0 := #sArrayInput[1, 47];
	    #sRecv.TeatTime.%B1 := #sArrayInput[1, 48];
	    #sRecv.TeatTime.%B2 := #sArrayInput[1, 49];
	    #sRecv.TeatTime.%B3 := #sArrayInput[1, 50];
	    #sRecv.DumpTime.%B0 := #sArrayInput[1, 53];
	    #sRecv.DumpTime.%B1 := #sArrayInput[1, 54];
	    #sRecv.DumpTime.%B2 := #sArrayInput[1, 55];
	    #sRecv.DumpTime.%B3 := #sArrayInput[1, 56];
	    
	    
	    
	    CASE #sRecv.LeakUnitCode OF
	        0000:
	            #sRecv.Result.Leak.Unit := 'cm3/s';
	        1000:
	            #sRecv.Result.Leak.Unit := 'cm3/min';
	        2000:
	            #sRecv.Result.Leak.Unit := 'cm3/h';
	        3000:
	            #sRecv.Result.Leak.Unit := 'mm3/h';
	        4000:
	            #sRecv.Result.Leak.Unit := 'Pa';
	        5000:
	            #sRecv.Result.Leak.Unit := 'Pa/s';
	        6000:
	            #sRecv.Result.Leak.Unit := 'Pa';
	        7000:
	            #sRecv.Result.Leak.Unit := 'Pa';
	        8000:
	            #sRecv.Result.Leak.Unit := 'Pa/s';
	        9000:
	            #sRecv.Result.Leak.Unit := 'Pa/s';
	        11000:
	            #sRecv.Result.Leak.Unit := 'bar';
	        12000:
	            #sRecv.Result.Leak.Unit := 'KPa';
	        13000:
	            #sRecv.Result.Leak.Unit := 'psi';
	        14000:
	            #sRecv.Result.Leak.Unit := 'mbar';
	        15000:
	            #sRecv.Result.Leak.Unit := 'MPa';
	        43000:
	            #sRecv.Result.Leak.Unit := 'Pa';
	        44000:
	            #sRecv.Result.Leak.Unit := 'Pa';
	        45000:
	            #sRecv.Result.Leak.Unit := 'Pa/s';
	        46000:
	            #sRecv.Result.Leak.Unit := 'In3/s';
	        47000:
	            #sRecv.Result.Leak.Unit := 'In3/min';
	        48000:
	            #sRecv.Result.Leak.Unit := 'In3/h';
	        49000:
	            #sRecv.Result.Leak.Unit := 'Ft3/h';
	        50000:
	            #sRecv.Result.Leak.Unit := 'mL/s';
	        51000:
	            #sRecv.Result.Leak.Unit := 'mL/min';
	        52000:
	            #sRecv.Result.Leak.Unit := 'mL/h';
	        58000:
	            #sRecv.Result.Leak.Unit := 'cm3/s';
	        59000:
	            #sRecv.Result.Leak.Unit := 'cm3/min';
	        60000:
	            #sRecv.Result.Leak.Unit := 'cm3/h';
	        76000:
	            #sRecv.Result.Leak.Unit := 'Ft3/s';
	        77000:
	            #sRecv.Result.Leak.Unit := 'Ft3/min';
	        84000:
	            #sRecv.Result.Leak.Unit := 'sccm';
	        ELSE
	            ;
	    END_CASE;
	    
	    (* detection mode change *)
	    IF NOT #iSysRun OR (#iManual XOR #sHelp.ManualOld) OR (#iAuto XOR #sHelp.AutoOld) THEN
	        #sHMI.Trigger.SetProg := FALSE;
	        #sHMI.Trigger.Measure := FALSE;
	        #ioSetProg := FALSE;
	        #ioMeasure := FALSE;
	        (* reset outputs *)
	        // Todo
	    END_IF;
	    #sHelp.ManualOld := #iManual;
	    #sHelp.AutoOld := #iAuto;
	    
	    (* detection rising edges of inputs *)
	    IF #iManual THEN
	        #ioSetProg := FALSE;
	        #ioMeasure := FALSE;
	    ELSIF #iAuto THEN
	        #sHMI.Trigger.SetProg := FALSE;
	        #sHMI.Trigger.Measure := FALSE;
	    END_IF;
	    #sHelp.ResetRis := NOT #sHelp.ResetOld AND #iReset;
	    #sHelp.ResetOld := #iReset;
	    #sHelp.SetProgRis := NOT #sHelp.SetProgOld AND (#sHMI.Trigger.SetProg OR #ioSetProg);
	    #sHelp.SetProgOld := #sHMI.Trigger.SetProg OR #ioSetProg;
	    #sHelp.MeasureRis := NOT #sHelp.MeasureOld AND (#sHMI.Trigger.Measure OR #ioMeasure);
	    #sHelp.MeasureOld := #sHMI.Trigger.Measure OR #ioMeasure;
	    
	    (* order handling *)
	    #sHelp.OrderCnt := 0;
	    IF #sHelp.SetProgOld THEN
	        #sHelp.OrderCnt := #sHelp.OrderCnt + 1;
	    END_IF;
	    IF #sHelp.MeasureOld THEN
	        #sHelp.OrderCnt := #sHelp.OrderCnt + 1;
	    END_IF;
	    IF (#sHelp.OrderCnt > 1) AND (#oErrorCode = 0) THEN
	        #oErrorCode := 201; // twice command request
	    END_IF;
	    IF (#oErrorCode = 0) AND NOT #oReady THEN
	        IF #sHelp.SetProgRis OR #sHelp.MeasureRis THEN
	            #oErrorCode := 200; // command while not ready
	        END_IF;
	    END_IF;
	    
	    (* error clear *)
	    IF (#sHelp.OrderCnt = 0) THEN
	        IF #sHelp.ResetRis THEN
	            #oErrorCode := 0;
	            #sSend.Reset := TRUE;
	        ELSE
	            #sSend.Reset := FALSE;
	        END_IF;
	    END_IF;
	    
	    (* check timeout *)
	    #sHelp.CmdTimer(IN := #sHelp.EnableTime,
	                    PT := #iTimeout);
	    (* Sequence --- SetProg *)
	    REGION SetProg
	        #tIndex := 1;
	        
	        IF (#oErrorCode = 0) AND #sHelp.SetProgRis THEN
	            #tZero := 0;
	            #tRetval.FILL := FILL(BVAL := #tZero, BLK => #oResult);
	            IF #iAuto THEN
	                #sHelp.Set := #sAuto.Set;
	            ELSE
	                #sHelp.Set := #sHMI.Set;
	            END_IF;
	            IF (#sHelp.Set.ProgNo >= 1) AND (#sHelp.Set.ProgNo <= 128) THEN
	                #sHelp.Abort := FALSE;
	                #sHelp.SetProgAct := TRUE;
	                #sHelp.Step[#tIndex] := 0;
	            ELSE
	                #oErrorCode := 202;
	            END_IF;
	        END_IF;
	        
	        IF NOT #sHelp.SetProgOld THEN
	            #oSetProgOk := FALSE;
	            IF #sHelp.SetProgAct THEN
	                #sHelp.Abort := TRUE;
	            END_IF;
	        END_IF;
	        
	        IF #sHelp.SetProgAct THEN
	            CASE #sHelp.Step[#tIndex] OF
	                0:  (* check error code *)
	                    IF #sRecv.ErrorCode <> 16#0000 THEN
	                        #sHelp.Step[#tIndex] := 1;
	                    ELSE
	                        #sHelp.Step[#tIndex] := 4;
	                    END_IF;
	                    
	                1:  (* start order *)
	                    IF #sRecv.Echo.Status = 16#0000 THEN
	                        #sSend.Reset := TRUE;
	                        #sHelp.EnableTime := FALSE;
	                        #sHelp.Step[#tIndex] := #sHelp.Step[#tIndex] + 1;
	                    END_IF;
	                    
	                2:  (* order accepted *)
	                    IF #sRecv.Echo.Reset AND #sRecv.ErrorCode = 16#FFFF THEN
	                        #sHelp.EnableTime := FALSE;
	                        #sHelp.Step[#tIndex] := #sHelp.Step[#tIndex] + 1;
	                    ELSE
	                        #sHelp.EnableTime := TRUE;
	                        IF #sHelp.CmdTimer.Q THEN
	                            #oErrorCode := 204;
	                            #sHelp.Step[#tIndex] := 99;
	                        END_IF;
	                    END_IF;
	                    
	                3:  (* order finished *)
	                    IF #sRecv.Echo.Reset AND #sRecv.ErrorCode <> 16#FFFF THEN
	                        #sSend.Reset := FALSE;
	                        #sHelp.EnableTime := FALSE;
	                        IF #sRecv.ErrorCode = 16#0000 THEN
	                            #sHelp.Step[#tIndex] := #sHelp.Step[#tIndex] + 1;
	                        ELSE
	                            #oErrorCode := 203;
	                            #sHelp.Step[#tIndex] := 99;
	                        END_IF;
	                    ELSE
	                        #sHelp.EnableTime := TRUE;
	                        IF #sHelp.CmdTimer.Q THEN
	                            #oErrorCode := 204;
	                            #sHelp.Step[#tIndex] := 99;
	                        END_IF;
	                    END_IF;
	                    
	                4:  (* start order *)
	                    IF (#sRecv.Echo.Status = 16#0000) THEN
	                        #sSend.ProgNo := #sHelp.Set.ProgNo - 1;
	                        #sSend.ProgramSel := TRUE;
	                        #sHelp.EnableTime := FALSE;
	                        #sHelp.Step[#tIndex] := #sHelp.Step[#tIndex] + 1;
	                    END_IF;
	                    
	                5:  (* order accepted *)
	                    IF #sRecv.Echo.ProgramSel AND #sRecv.ErrorCode = 16#FFFF THEN
	                        #sHelp.EnableTime := FALSE;
	                        #sHelp.Step[#tIndex] := #sHelp.Step[#tIndex] + 1;
	                    ELSE
	                        #sHelp.EnableTime := TRUE;
	                        IF #sHelp.CmdTimer.Q THEN
	                            #oErrorCode := 204;
	                            #sHelp.Step[#tIndex] := 995;
	                        END_IF;
	                    END_IF;
	                    
	                6:  (* order finished *)
	                    IF #sRecv.Echo.ProgramSel AND #sRecv.ErrorCode <> 16#FFFF THEN
	                        #sSend.ProgramSel := FALSE;
	                        #sHelp.EnableTime := FALSE;
	                        IF #sRecv.ErrorCode = 16#0000 THEN
	                            #sHelp.Step[#tIndex] := 996;
	                        ELSE
	                            #oErrorCode := 203;
	                            #sHelp.Step[#tIndex] := 997;
	                        END_IF;
	                    ELSE
	                        #sHelp.EnableTime := TRUE;
	                        IF #sHelp.CmdTimer.Q THEN
	                            #oErrorCode := 204;
	                            #sHelp.Step[#tIndex] := 998;
	                        END_IF;
	                    END_IF;
	                    
	                99,995,996,997,998,999:
	                    #sSend.Reset := FALSE;
	                    #sSend.ProgramSel := FALSE;
	                    #sHelp.SetProgAct := FALSE;
	                    #sHMI.Trigger.SetProg := FALSE;
	                    #sHelp.Abort := FALSE;
	                    IF #oErrorCode = 0 THEN
	                        #oSetProgOk := TRUE;
	                    END_IF;
	            END_CASE;
	        END_IF;
	    END_REGION
	    (* Sequence --- Measure *)
	    REGION Measure
	        #tIndex := 2;
	        
	        IF (#oErrorCode = 0) AND #sHelp.MeasureRis THEN
	            #tZero := 0;
	            #tRetval.FILL := FILL(BVAL := #tZero, BLK => #oResult);
	            IF #iAuto THEN
	                #sHelp.Set := #sAuto.Set;
	            ELSE
	                #sHelp.Set := #sHMI.Set;
	            END_IF;
	            #sHelp.Abort := FALSE;
	            #sHelp.MeasureAct := TRUE;
	            #sHelp.Step[#tIndex] := 0;
	        END_IF;
	        
	        IF NOT #sHelp.MeasureOld THEN
	            #oMeasureOk := FALSE;
	            IF #sHelp.MeasureAct THEN
	                #sHelp.Abort := TRUE;
	            END_IF;
	        END_IF;
	        
	        IF #sHelp.MeasureAct THEN
	            CASE #sHelp.Step[#tIndex] OF
	                0:  (* check error code *)
	                    IF #sRecv.ErrorCode <> 16#0000 THEN
	                        #sHelp.Step[#tIndex] := 1;
	                    ELSE
	                        #sHelp.Step[#tIndex] := 4;
	                    END_IF;
	                    
	                1:  (* start order *)
	                    IF #sRecv.Echo.Status = 16#0000 THEN
	                        #sSend.Reset := TRUE;
	                        #sHelp.EnableTime := FALSE;
	                        #sHelp.Step[#tIndex] := #sHelp.Step[#tIndex] + 1;
	                    END_IF;
	                    
	                2:  (* order accepted *)
	                    IF #sRecv.Echo.Reset AND #sRecv.ErrorCode = 16#FFFF THEN
	                        #sHelp.EnableTime := FALSE;
	                        #sHelp.Step[#tIndex] := #sHelp.Step[#tIndex] + 1;
	                    ELSE
	                        #sHelp.EnableTime := TRUE;
	                        IF #sHelp.CmdTimer.Q THEN
	                            #oErrorCode := 204;
	                            #sHelp.Step[#tIndex] := 299;
	                        END_IF;
	                    END_IF;
	                    
	                3:  (* order finished *)
	                    IF #sRecv.Echo.Reset AND #sRecv.ErrorCode <> 16#FFFF THEN
	                        #sSend.Reset := FALSE;
	                        #sHelp.EnableTime := FALSE;
	                        IF #sRecv.ErrorCode = 16#0000 THEN
	                            #sHelp.Step[#tIndex] := #sHelp.Step[#tIndex] + 1;
	                        ELSE
	                            #oErrorCode := 203;
	                            #sHelp.Step[#tIndex] := 398;
	                        END_IF;
	                    ELSE
	                        #sHelp.EnableTime := TRUE;
	                        IF #sHelp.CmdTimer.Q THEN
	                            #oErrorCode := 204;
	                            #sHelp.Step[#tIndex] := 399;
	                        END_IF;
	                    END_IF;
	                    
	                4:  (* start order *)
	                    IF (#sRecv.Echo.Status = 16#0000) THEN
	                        #sSend.Start := TRUE;
	                        #sHelp.EnableTime := FALSE;
	                        #sHelp.Step[#tIndex] := #sHelp.Step[#tIndex] + 1;
	                    END_IF;
	                    
	                5:  (* order accepted *)
	                    IF #sRecv.Echo.Start AND #sRecv.ErrorCode = 16#FFFF THEN
	                        #sHelp.EnableTime := FALSE;
	                        #sHelp.Step[#tIndex] := #sHelp.Step[#tIndex] + 1;
	                    ELSE
	                        #sHelp.EnableTime := TRUE;
	                        IF #sHelp.CmdTimer.Q THEN
	                            #oErrorCode := 204;
	                            #sHelp.Step[#tIndex] := 599;
	                        END_IF;
	                    END_IF;
	                    
	                6:  (* order finished *)
	                    IF #sRecv.Echo.Start AND #sRecv.ErrorCode <> 16#FFFF THEN
	                        #sSend.Start := FALSE;
	                        #sHelp.EnableTime := FALSE;
	                        IF #sRecv.ErrorCode = 16#0000 THEN
	                            #sHelp.Step[#tIndex] := #sHelp.Step[#tIndex] + 1;
	                        ELSE
	                            #oErrorCode := 203;
	                            #sHelp.Step[#tIndex] := 698;
	                        END_IF;
	                    ELSIF #sHelp.Abort THEN
	                        #sHelp.Step[#tIndex] := 10;
	                    ELSE
	                        #sHelp.EnableTime := TRUE;
	                        IF #sHelp.CmdTimer.Q THEN
	                            #oErrorCode := 204;
	                            #sHelp.Step[#tIndex] := 699;
	                        END_IF;
	                    END_IF;
	                    
	                7:  (* start order *)
	                    IF (#sRecv.Echo.Status = 16#0000) AND #sRecv.CycleEnd THEN
	                        #sSend.ReadLastResult := TRUE;
	                        #sHelp.EnableTime := FALSE;
	                        #sHelp.Step[#tIndex] := #sHelp.Step[#tIndex] + 1;
	                    END_IF;
	                    
	                8:  (* order accepted *)
	                    IF #sRecv.Echo.ReadLastResult AND #sRecv.ErrorCode = 16#FFFF THEN
	                        #sHelp.EnableTime := FALSE;
	                        #sHelp.Step[#tIndex] := #sHelp.Step[#tIndex] + 1;
	                    ELSE
	                        #sHelp.EnableTime := TRUE;
	                        IF #sHelp.CmdTimer.Q THEN
	                            #oErrorCode := 204;
	                            #sHelp.Step[#tIndex] := 899;
	                        END_IF;
	                    END_IF;
	                    
	                9:  (* order finished *)
	                    IF #sRecv.Echo.ReadLastResult AND #sRecv.ErrorCode <> 16#FFFF THEN
	                        #sSend.ReadLastResult := FALSE;
	                        #sHelp.EnableTime := FALSE;
	                        IF #sRecv.ErrorCode = 16#0000 THEN
	                            #sHelp.Step[#tIndex] := 997;
	                        ELSE
	                            #oErrorCode := 203;
	                            #sHelp.Step[#tIndex] := 998;
	                        END_IF;
	                    ELSE
	                        #sHelp.EnableTime := TRUE;
	                        IF #sHelp.CmdTimer.Q THEN
	                            #oErrorCode := 204;
	                            #sHelp.Step[#tIndex] := 999;
	                        END_IF;
	                    END_IF;
	                    
	                10:  (* abort order *)
	                    #sHelp.Step[#tIndex] := 1099;
	                    
	                299,398,399,599,698,699,899,997,998,999,1099:
	                    #sSend.Reset := FALSE;
	                    #sSend.Start := FALSE;
	                    #sSend.ReadLastResult := FALSE;
	                    #sHelp.MeasureAct := FALSE;
	                    #sHMI.Trigger.Measure := FALSE;
	                    #sHelp.Abort := FALSE;
	                    IF #oErrorCode = 0 THEN
	                        #oResult := #sRecv.Result;
	                        #oMeasureOk := TRUE;
	                    END_IF;
	            END_CASE;
	        END_IF;
	    END_REGION
	    
	    (* update outputs *)
	    #oDeviceReady := #sRecv.CycleEnd;
	    #oPressure.Value := UDINT_TO_REAL(#sRecv.ActPressure) / 1000.0;
	    CASE #sRecv.PressureUnitCode OF
	        0000:
	            #oPressure.Unit := 'cm3/s';
	        1000:
	            #oPressure.Unit := 'cm3/min';
	        2000:
	            #oPressure.Unit := 'cm3/h';
	        3000:
	            #oPressure.Unit := 'mm3/h';
	        4000:
	            #oPressure.Unit := 'Pa';
	        5000:
	            #oPressure.Unit := 'Pa/s';
	        6000:
	            #oPressure.Unit := 'Pa';
	        7000:
	            #oPressure.Unit := 'Pa';
	        8000:
	            #oPressure.Unit := 'Pa/s';
	        9000:
	            #oPressure.Unit := 'Pa/s';
	        11000:
	            #oPressure.Unit := 'bar';
	        12000:
	            #oPressure.Unit := 'KPa';
	        13000:
	            #oPressure.Unit := 'psi';
	        14000:
	            #oPressure.Unit := 'mbar';
	        15000:
	            #oPressure.Unit := 'MPa';
	        43000:
	            #oPressure.Unit := 'Pa';
	        44000:
	            #oPressure.Unit := 'Pa';
	        45000:
	            #oPressure.Unit := 'Pa/s';
	        46000:
	            #oPressure.Unit := 'In3/s';
	        47000:
	            #oPressure.Unit := 'In3/min';
	        48000:
	            #oPressure.Unit := 'In3/h';
	        49000:
	            #oPressure.Unit := 'Ft3/h';
	        50000:
	            #oPressure.Unit := 'mL/s';
	        51000:
	            #oPressure.Unit := 'mL/min';
	        52000:
	            #oPressure.Unit := 'mL/h';
	        58000:
	            #oPressure.Unit := 'cm3/s';
	        59000:
	            #oPressure.Unit := 'cm3/min';
	        60000:
	            #oPressure.Unit := 'cm3/h';
	        76000:
	            #oPressure.Unit := 'Ft3/s';
	        77000:
	            #oPressure.Unit := 'Ft3/min';
	        84000:
	            #oPressure.Unit := 'sccm';
	        ELSE
	            ;
	    END_CASE;
	    #oActProgStep := #sRecv.ActProgStep;
	    #oActProgNo := #sRecv.ActProgram + 1;
	    
	    (* update hmi *)
	    #sHMI.Status.DeviceReady := #oDeviceReady;
	    #sHMI.Status.Ready := #oReady;
	    #sHMI.Status.Error := #oError;
	    #sHMI.Status.SetProgOk := #oSetProgOk;
	    #sHMI.Status.MeasureOk := #oMeasureOk;
	    #sHMI.Status.ErrorCode := #oErrorCode;
	    #sHMI.Status.Result := #oResult;
	    #sHMI.Status.Pressure := #oPressure;
	    #sHMI.Status.ActProgStep := #oActProgStep;
	    #sHMI.Status.ActProgNo := #oActProgNo;
	    #sHMI.Status.ElapsedTime := #oElapsedTime;
	    
	    (* set ready for command flag *)
	    IF (#oErrorCode = 0) AND (#sHelp.OrderCnt = 0) AND #oDeviceReady AND NOT #sHelp.SetProgAct AND NOT #sHelp.MeasureAct THEN
	        #oReady := TRUE;
	    ELSE
	        #oReady := FALSE;
	    END_IF;
	    
	    (* move static bits to output bytes *)
	    #sArrayOutput[1, 1].%X0 := #sSend.Reset;
	    #sArrayOutput[1, 1].%X1 := #sSend.Start;
	    #sArrayOutput[1, 1].%X2 := #sSend.StartSpec;
	    #sArrayOutput[1, 1].%X3 := #sSend.ProgramSel AND "ClockMemory0.8s";
	    #sArrayOutput[1, 1].%X5 := #sSend.ReadPara ;
	    #sArrayOutput[1, 2].%X7 := #sSend.ReadLastResult AND "ClockMemory0.8s";
	    #sArrayOutput[1, 7] := #sSend.ProgNo.%B0;
	    REGION SpecialCycle
	        // Statement section REGION
	        IF NOT #ioSpecialCycle THEN
	            #SpecialCycleStep := 0;
	        END_IF;
	        IF #ioSpecialCycle AND #SpecialCycleStep = 0 AND #oReady AND #oDeviceReady THEN
	            #SpecialCycleStep := 10;
	        END_IF;
	        #IEC_Timer_0_Instance(IN := #SpecialCycleStep = 10,
	                              PT := t#0.2s);
	        #IEC_Timer_1_Instance(IN := #SpecialCycleStep = 20,
	                              PT := t#0.4s);
	        CASE #SpecialCycleStep OF
	            10://标志清零
	                #sHelp.EnableTime := FALSE;
	                #sArrayOutput[1, 9] := 16#00;
	                #sArrayOutput[1, 10] := 16#00;
	                IF #IEC_Timer_0_Instance.Q THEN
	                    #SpecialCycleStep := 20;
	                END_IF;
	            20://赋值
	                #sHelp.EnableTime := FALSE;
	                #sArrayOutput[1, 9] := 16#08;
	                #sArrayOutput[1, 10] := 16#00;
	                #sSend.StartSpec := 1;
	                IF #IEC_Timer_1_Instance.Q THEN
	                    #SpecialCycleStep := 30;
	                END_IF;
	                
	            30://触发
	                #sHelp.EnableTime := FALSE;
	                #sSend.Start := 1;
	                #SpecialCycleStep := 40;
	            40://运行
	                IF #sRecv.Echo.StartSpec THEN
	                    #sHelp.EnableTime := FALSE;
	                    #SpecialCycleStep := 50;
	                END_IF;
	                #sHelp.EnableTime := TRUE;
	                IF #sHelp.CmdTimer.Q THEN
	                    #oErrorCode := 1004;
	                    #SpecialCycleStep := 99;
	                END_IF;
	            50://完成
	                IF NOT #oReady AND NOT #oDeviceReady THEN
	                    #sHelp.EnableTime := FALSE;
	                    #sSend.Start := #sSend.StartSpec := 0;
	                    #SpecialCycleStep := 60;
	                END_IF;
	                #sHelp.EnableTime := TRUE;
	                IF #sHelp.CmdTimer.Q THEN
	                    #oErrorCode := 1005;
	                    #SpecialCycleStep := 99;
	                END_IF;
	            60://完成
	                IF #oReady AND #oDeviceReady THEN
	                    #ioSpecialCycle := #sSend.StartSpec := 0;
	                    #sHelp.EnableTime := FALSE;
	                END_IF;
	            99:
	                #sSend.Start := #sSend.StartSpec := 0;
	                #ioSpecialCycle := 0;
	        END_CASE;
	        
	    END_REGION
	    REGION ReadProTime
	        // Statement section REGION
	        IF NOT #ioReadProTime THEN
	            #ReadProTimeStep := 0;
	        END_IF;
	        IF #ioReadProTime AND #ReadProTimeStep = 0 AND #oReady AND #oDeviceReady THEN
	            #ReadProTimeStep := 10;
	        END_IF;
	        #IEC_Timer_0_Instance_1(IN := #ReadProTimeStep = 20,
	                              PT := t#0.1s);
	      #IEC_Timer_1_Instance_1(IN := #ReadProTimeStep = 20,
	                              PT := t#0.3s);
	      
	        CASE #ReadProTimeStep OF
	            10://标志
	                #sHelp.EnableTime := FALSE;
	                #sArrayOutput[1, 33] := 16#04;
	                #sArrayOutput[1, 34] := 16#00;
	                #sArrayOutput[1, 35] := 16#01;
	                #sArrayOutput[1, 36] := 16#00;
	                #sArrayOutput[1, 37] := 16#02;
	                #sArrayOutput[1, 38] := 16#00;
	                #sArrayOutput[1, 39] := 16#03;
	                #sArrayOutput[1, 40] := 16#00;
	                #sArrayOutput[1, 41] := 16#09;
	                #sArrayOutput[1, 42] := 16#00;
	                #ReadProTimeStep := 20;
	                
	            20://赋值
	                #sHelp.EnableTime := FALSE;
	                #sArrayOutput[1, 33] := 16#04;
	                #sArrayOutput[1, 34] := 16#00;
	                #sArrayOutput[1, 35] := 16#01;
	                #sArrayOutput[1, 36] := 16#00;
	                #sArrayOutput[1, 37] := 16#02;
	                #sArrayOutput[1, 38] := 16#00;
	                #sArrayOutput[1, 39] := 16#03;
	                #sArrayOutput[1, 40] := 16#00;
	                #sArrayOutput[1, 41] := 16#09;
	                #sArrayOutput[1, 42] := 16#00;
	                
	                IF #IEC_Timer_0_Instance_1.Q THEN
	                    #sSend.ReadPara := 1;
	                END_IF;
	                IF  #sRecv.Echo.ReadPara OR #IEC_Timer_1_Instance_1.Q THEN
	                    #ReadProTimeStep := 30;
	                END_IF;
	            30://触发
	                #sHelp.EnableTime := FALSE;
	               
	                #ReadProTimeStep := 40;
	            40://运行
	                #ReadProTimeStep := 50;
	                #sHelp.EnableTime := TRUE;
	                IF #sHelp.CmdTimer.Q THEN 
	                    #oErrorCode := 1004;
	                    #ReadProTimeStep := 99;
	                END_IF;
	            50://完成
	                #ReadProTimeStep := 60;
	                
	            60://完成
	                IF #oReady AND #oDeviceReady THEN
	                    #ioReadProTime := #sSend.ReadPara := 0;
	                    #sHelp.EnableTime := FALSE;
	                END_IF;
	            99:
	                #sSend.Start := #sSend.ReadPara := 0;
	                #ioReadProTime := 0;
	        END_CASE;
	        
	    END_REGION
	
	    
	    (* Cyclic write plc output to tester input *)
	    #tRetval.DPWR[1] := DPWR_DAT(LADDR := #iHWID_Slot5,
	                                 RECORD := #sArrayOutput[1]);
	    #tRetval.DPWR[2] := DPWR_DAT(LADDR := #iHWID_Slot6,
	                                 RECORD := #sArrayOutput[2]);
	    #tRetval.DPWR[3] := DPWR_DAT(LADDR := #iHWID_Slot7,
	                                 RECORD := #sArrayOutput[3]);
	    #tRetval.DPWR[4] := DPWR_DAT(LADDR := #iHWID_Slot8,
	                                 RECORD := #sArrayOutput[4]);
	    IF #tRetval.DPWR[1] <> 0 OR
	        #tRetval.DPWR[2] <> 0 OR
	        #tRetval.DPWR[3] <> 0 OR
	        #tRetval.DPWR[4] <> 0  THEN
	        #oErrorCode := 101; // Error cyclic write
	    END_IF;
	    
	    (* handle errors within block *)
	    #tRetval.LocallyErrID := GET_ERR_ID();
	    IF #tRetval.LocallyErrID <> 0 THEN
	        (* reset fieldbus output *)
	        FOR #tLoop := 1 TO UINT_TO_INT(#cSlotAmount) DO
	            UFILL_BLK(IN := 0,
	                      COUNT := #cFieldbusBytes,
	                      OUT => #sArrayOutput[#tLoop, 01]);
	        END_FOR;
	        #oErrorCode := 102; // Error within block
	    END_IF;
	    
	END_IF;
END_FUNCTION_BLOCK

FUNCTION_BLOCK "DT-Chars"
{ S7_Optimized_Access := 'FALSE' }
VERSION : 0.1
   VAR_INPUT 
      YEAR : Int;
      MONTH : Int;
      DAY : Int;
      HH : Int;
      MM : Int;
      SS : Int;
   END_VAR

   VAR_OUTPUT 
      Year_Byte1 : Char;
      Year_Byte2 : Char;
      Month_Byte1 : Char;
      Month_Byte2 : Char;
      Days_Byte1 : Char;
      Days_Byte2 : Char;
      HH_Byte1 : Char;
      HH_Byte2 : Char;
      MM_Byte1 : Char;
      MM_Byte2 : Char;
      SS_Byte1 : Char;
      SS_Byte2 : Char;
      CalculateDays_Byte1 : Char;
      CalculateDays_Byte2 : Char;
      CalculateDays_Byte3 : Char;
      Error_Code : Int;
      Year_Byte3 : String[1];
      Year_Byte4 : String[1];
      Month_Byte3 : String[1];
      Month_Byte4 : String[1];
      Days_Byte3 : String[1];
      Days_Byte4 : String[1];
      HH_Byte3 : String[1];
      HH_Byte4 : String[1];
      MM_Byte3 : String[1];
      MM_Byte4 : String[1];
      SS_Byte3 : String[1];
      SS_Byte4 : String[1];
      CalculateDays_Byte4 : String[1];
      CalculateDays_Byte5 : String[1];
      CalculateDays_Byte6 : String[1];
      OTimeStr : String[20];
   END_VAR

   VAR 
      Sum_Days : Int;
      Sum_Year : Int;
   END_VAR

   VAR_TEMP 
      Input_1_BCD : Word;
      Input_2_BCD : Word;
      Input_3_BCD : Word;
      Input_4_BCD : Word;
      Input_5_BCD : Word;
      Input_6_BCD : Word;
      Input_7_BCD : Word;
   END_VAR


BEGIN
	#Input_1_BCD := INT_TO_BCD16(#YEAR);
	#Year_Byte2 := INT_TO_BYTE(#YEAR MOD 10 + 48);
	#Year_Byte1 := INT_TO_BYTE(WORD_TO_INT(SHR(IN := #Input_1_BCD, N := 4)) + 48);
	
	
	#Input_2_BCD := INT_TO_BCD16(#MONTH);
	#Month_Byte2 := INT_TO_BYTE(#MONTH MOD 10 + 48);
	#Month_Byte1 := INT_TO_BYTE(WORD_TO_INT(SHR(IN := #Input_2_BCD, N := 4)) + 48);
	
	#Input_3_BCD := INT_TO_BCD16(#DAY);
	#Days_Byte2 := INT_TO_BYTE(#DAY MOD 10 + 48);
	#Days_Byte1 := INT_TO_BYTE(WORD_TO_INT(SHR(IN := #Input_3_BCD, N := 4)) + 48);
	
	#Input_4_BCD := INT_TO_BCD16(#HH);
	#HH_Byte2 := INT_TO_BYTE(#HH MOD 10 + 48);
	#HH_Byte1 := INT_TO_BYTE(WORD_TO_INT(SHR(IN := #Input_4_BCD, N := 4)) + 48);
	
	#Input_5_BCD := INT_TO_BCD16(#MM);
	#MM_Byte2 := INT_TO_BYTE(#MM MOD 10 + 48);
	#MM_Byte1 := INT_TO_BYTE(WORD_TO_INT(SHR(IN := #Input_5_BCD, N := 4)) + 48);
	
	#Input_6_BCD := INT_TO_BCD16(#SS);
	#SS_Byte2 := INT_TO_BYTE(#SS MOD 10 + 48);
	#SS_Byte1 := INT_TO_BYTE(WORD_TO_INT(SHR(IN := #Input_6_BCD, N := 4)) + 48);
	
	#Sum_Days := 0;//初始值
	#Sum_Year := 2000 + #YEAR;
	CASE #MONTH OF
	    12:
	        #Sum_Days := 31 + 28 + 31 + 30 + 31 + 30 + 31 + 31 + 30 + 31 + 30 + #DAY;
	    11:
	        #Sum_Days := 31 + 28 + 31 + 30 + 31 + 30 + 31 + 31 + 30 + 31 + #DAY;
	    10:
	        #Sum_Days := 31 + 28 + 31 + 30 + 31 + 30 + 31 + 31 + 30 + #DAY;
	    9:
	        #Sum_Days := 31 + 28 + 31 + 30 + 31 + 30 + 31 + 31 + #DAY;
	    8:
	        #Sum_Days := 31 + 28 + 31 + 30 + 31 + 30 + 31 + #DAY;
	    7:
	        #Sum_Days := 31 + 28 + 31 + 30 + 31 + 30 + #DAY;
	    6:
	        #Sum_Days := 31 + 28 + 31 + 30 + 31 + #DAY;
	    5:
	        #Sum_Days := 31 + 28 + 31 + 30 + #DAY;
	    4:
	        #Sum_Days := 31 + 28 + 31 + #DAY;
	    3:
	        #Sum_Days := 31 + 28 + #DAY;
	    2:
	        #Sum_Days := 31 + #DAY;
	    1:
	        #Sum_Days := #DAY;
	
	END_CASE;
	
	//判断是否是闰年 闰年2月29天
	IF (#Sum_Year MOD 4=0)AND(#Sum_Year MOD 100<>0)OR(#Sum_Year MOD 400=0)AND(#MONTH > 2) THEN
	        // Statement section IF 
	    #Sum_Days := #Sum_Days +1;//闰年2月+1    
	END_IF;
	
	#Input_4_BCD:=INT_TO_BCD16(#Sum_Days);
	#CalculateDays_Byte3 := INT_TO_BYTE(WORD_TO_INT(SHR(IN := (#Input_4_BCD AND 16#000F), N :=0 )) + 48);
	#CalculateDays_Byte2 := INT_TO_BYTE(WORD_TO_INT(SHR(IN := (#Input_4_BCD AND 16#00F0), N := 4)) + 48);
	#CalculateDays_Byte1 := INT_TO_BYTE(WORD_TO_INT(SHR(IN := (#Input_4_BCD AND 16#0F00), N := 8)) + 48);
	
	#Year_Byte3 := CHAR_TO_STRING(#Year_Byte1);
	#Year_Byte4 := CHAR_TO_STRING(#Year_Byte2);
	
	#Month_Byte3 := CHAR_TO_STRING(#Month_Byte1);
	#Month_Byte4 := CHAR_TO_STRING(#Month_Byte2);
	
	#Days_Byte3 := CHAR_TO_STRING(#Days_Byte1);
	#Days_Byte4 := CHAR_TO_STRING(#Days_Byte2);
	
	#HH_Byte3 := CHAR_TO_STRING(#HH_Byte1);
	#HH_Byte4 := CHAR_TO_STRING(#HH_Byte2);
	
	#MM_Byte3 := CHAR_TO_STRING(#MM_Byte1);
	#MM_Byte4 := CHAR_TO_STRING(#MM_Byte2);
	
	#SS_Byte3 := CHAR_TO_STRING(#SS_Byte1);
	#SS_Byte4 := CHAR_TO_STRING(#SS_Byte2);
	
	#CalculateDays_Byte4 := CHAR_TO_STRING(#CalculateDays_Byte1);
	#CalculateDays_Byte5 := CHAR_TO_STRING(#CalculateDays_Byte2);
	#CalculateDays_Byte6 := CHAR_TO_STRING(#CalculateDays_Byte3);
	
	
	#OTimeStr := CONCAT(IN1 := '20', IN2 := #Year_Byte3, IN3 := #Year_Byte4, IN4 := '-',
	                                 IN5 := #Month_Byte3, IN6 := #Month_Byte4, IN7 := '-',
	                                 IN8 := #Days_Byte3, IN9 := #Days_Byte4, IN10 := ' ',
	                                 IN11 := #HH_Byte3, IN12 := #HH_Byte4, IN13 := ':',
	                                 IN14 := #MM_Byte3, IN15 := #MM_Byte4, IN16 := ':',
	                                 IN17 := #SS_Byte3, IN18 := #SS_Byte4);
	
	
	
	
	
END_FUNCTION_BLOCK

FUNCTION_BLOCK "FB_KeyenceCheckerIV3"
{ S7_Optimized_Access := 'TRUE' }
VERSION : 0.1
   VAR_INPUT 
      I_nID : Int;
   END_VAR

   VAR 
      rtrigManualMode {InstructionName := 'R_TRIG'; LibVersion := '1.0'} : R_TRIG;
      ftrigManualMode {InstructionName := 'F_TRIG'; LibVersion := '1.0'} : F_TRIG;
      "****Common*******" : Bool;
      nStep : Int;
      nNextStep : Int;
      nLastStep : Int;
      bCondition : Bool;
      fbNextstep { S7_SetPoint := 'False'} : "FB_Next";
      tonProcessOvertime {InstructionName := 'TON_TIME'; LibVersion := '1.0'; S7_SetPoint := 'False'} : TON_TIME;
      "****Local******" : Bool;
      aToolResultReset : Array[1..64] of Bool;
      ToolResultResult : Array[1..64] of Struct
         nToolMatchingRate : Word;
         nToolMatchingRateMAX : Word;
         nToolMatchingRateMIN : Word;
         nToolLowerLimitValue : Word;
         nToolUpperLimitValue : Word;
         nDecimalPosition : Word;
         "nPitchPresentValueMAX/ColorAverageH (hue)" : Word;
         "nPitchPresentValueMIN/ColorAverageS(saturation)" : Word;
         "nNumberOfPitches/ColorAverageV(brightness)/BrightnessAverage" : Word;
         nReserved1 : Word;
      END_STRUCT;
      bCompleteToggleSign : Bool;
      rtrigCompleteToggle {InstructionName := 'R_TRIG'; LibVersion := '1.0'; S7_SetPoint := 'False'} : R_TRIG;
      ftrigCompleteToggle {InstructionName := 'F_TRIG'; LibVersion := '1.0'; S7_SetPoint := 'False'} : F_TRIG;
      nIdx : Int;
      nTriggerFailCount : Byte;
      "****Instruction******" : Bool;
   END_VAR
   VAR DB_SPECIFIC
      nWord : Word;
      aWord { ExternalAccessible := 'False'; ExternalVisible := 'False'; ExternalWritable := 'False'} AT nWord : Array[0..1] of Byte;
      nDWord : DWord;
      aDWord { ExternalAccessible := 'False'; ExternalVisible := 'False'; ExternalWritable := 'False'} AT nDWord : Array[0..3] of Byte;
   END_VAR
   VAR 
      nIndex3 : Int;
   END_VAR

   VAR_TEMP 
      nByte : Byte;
      aInput_Byte1 : Array[0..3] of Byte;
      aInput_Byte2 : Array[0..3] of Byte;
      aInput_Byte3 : Array[0..15] of Byte;
      aInput_Byte4 : Array[0..27] of Byte;
      aInput_Byte5 : Array[0..19] of Byte;
      aInput_Byte6 : Array[0..63] of Struct
         bInput_Byte0 : Byte;
         bInput_Byte1 : Byte;
         bInput_Byte2 : Byte;
         bInput_Byte3 : Byte;
         bInput_Byte4 : Byte;
         bInput_Byte5 : Byte;
         bInput_Byte6 : Byte;
         bInput_Byte7 : Byte;
         bInput_Byte8 : Byte;
         bInput_Byte9 : Byte;
         bInput_Byte10 : Byte;
         bInput_Byte11 : Byte;
         bInput_Byte12 : Byte;
         bInput_Byte13 : Byte;
         bInput_Byte14 : Byte;
         bInput_Byte15 : Byte;
         bInput_Byte16 : Byte;
         bInput_Byte17 : Byte;
         bInput_Byte18 : Byte;
         bInput_Byte19 : Byte;
      END_STRUCT;
      aInput_Byte7 : Array[0..7] of Byte;
      aOutput_Byte1 : Array[0..11] of Byte;
      aRetvalRead : Array[1..22] of Int;
      aRetvalWrite : Array[1..1] of Int;
   END_VAR

   VAR CONSTANT 
      MODE_CHECKER_IDLE : Int := 0;
      MODE_CHECKER_START : Int := 1;
      MODE_CHECKER_REGISTER : Int := 4;
      MODE_CHECKER_CLEAR : Int := 5;
      MODE_CHECKER_RESET : Int := 99;
   END_VAR


BEGIN
	(*
	=============================================================================
	BBSS Automation
	(c)Copyright 2022 All Rights Reserved
	-----------------------------------------------------------------------------
	Functionality:
	This function block manager keyence checker iv3 control
	-----------------------------------------------------------------------------
	Change log table:
	Version   Date Y/M/D    Person       Description
	3.0.1     21/09/01      Xiangxiang   Active simulation
	3.0.4     22/01/20      Yuan Li      Handshake disabled
	3.0.5     22/05/13      Xuecao Guo   Update IV2 to IV3
	4.0.0     22/08/18      Huiyun       Separate condition and definition
	=============================================================================
	*)
	
